      A     M   1503.7;
      A     M    184.1;
      A     M   1606.6;
      A     M   1600.0;
      O     ;
      A     M   1503.5;
      A     M    184.0;
      A(    ;
      O     M   1707.0;
      O     ;
      A     M   1702.0;
      A     M   1702.2;
      A     M   1702.4;
      A     M   1702.6;
      A     M   1703.0;
      A     M   1703.2;
      A     M   1703.4;
      A     M   1703.6;
      A     M   1706.7;
      A     M   1704.0;
      A     M   1704.2;
      A     M   1704.5;
      A     M   1704.6;
      )     ;
      A     M   1706.1;
      A     M   1701.0;
      =     Q   1058.0;
NETWORK
TITLE =

      A     M   4108.1;
      =     Q   1058.1;
NETWORK
TITLE =

      A     M   1503.7;
      A     M    184.1;
      A     M   1606.6;
      A     M   1600.0;
      =     Q   1059.0;
NETWORK
TITLE =

      A     M   1503.5;
      A     M    184.0;
      A     M   1701.0;
      A     M   1706.1;
      A(    ;
      O     M   1707.0;
      O     ;
      A     M   1702.0;
      A     M   1702.2;
      A     M   1702.4;
      A     M   1702.6;
      A     M   1703.0;
      A     M   1703.2;
      A     M   1703.4;
      A     M   1703.6;
      A     M   1706.7;
      A     M   1704.0;
      A     M   1704.2;
      A     M   1704.5;
      A     M   1704.6;
      )     ;
      =     Q   1059.2;
END_FUNCTION

FUNCTION FC 137 : VOID
TITLE =
VERSION : 0.1

BEGIN
NETWORK
TITLE =
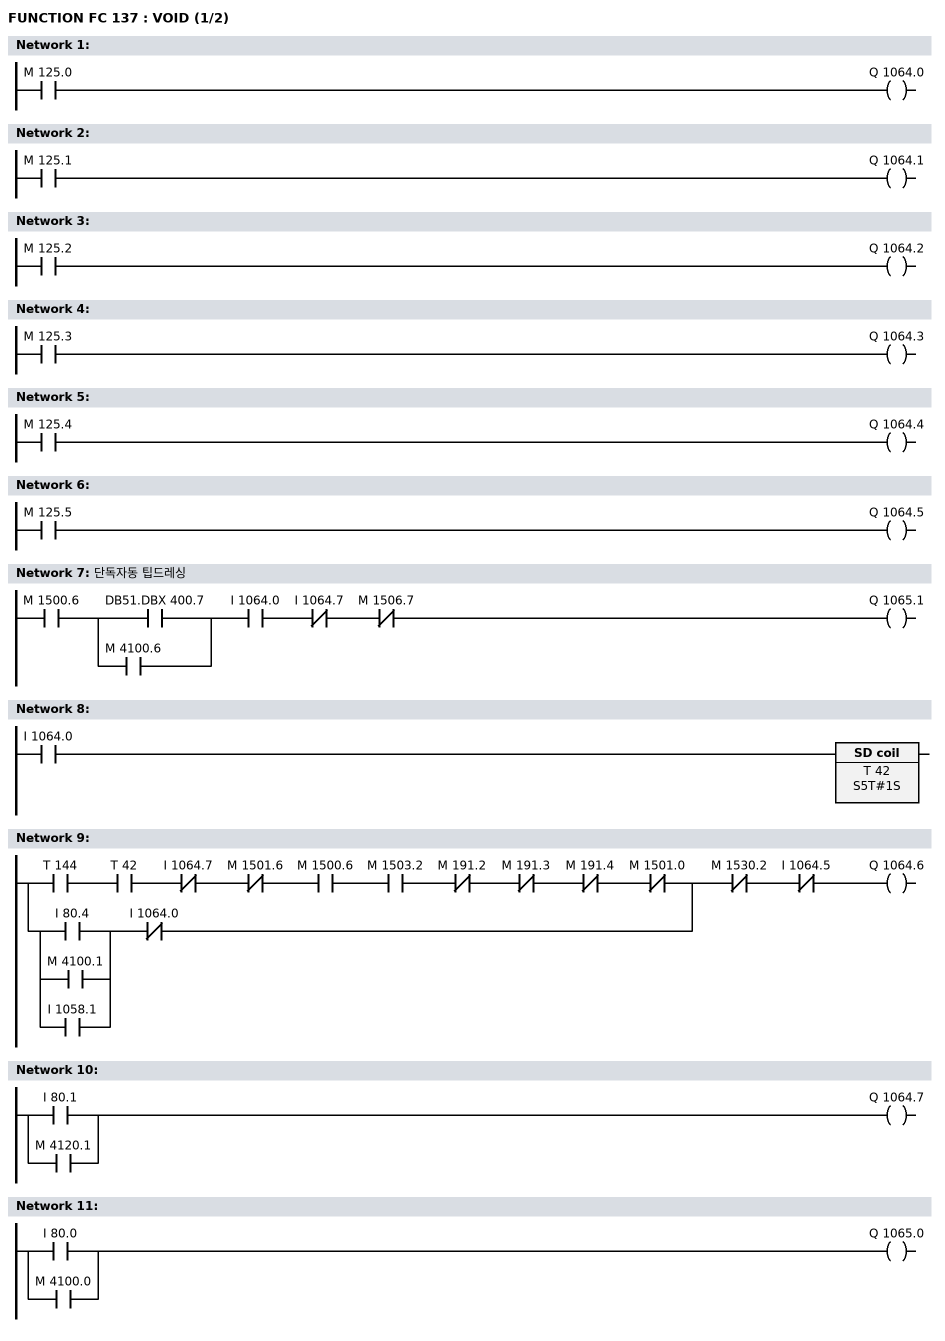

      A     M    125.0;
      =     Q   1064.0;
NETWORK
TITLE =

      A     M    125.1;
      =     Q   1064.1;
NETWORK
TITLE =

      A     M    125.2;
      =     Q   1064.2;
NETWORK
TITLE =

      A     M    125.3;
      =     Q   1064.3;
NETWORK
TITLE =

      A     M    125.4;
      =     Q   1064.4;
NETWORK
TITLE =

      A     M    125.5;
      =     Q   1064.5;
NETWORK
TITLE =단독자동 팁드레싱

      A     M   1500.6;
      A(    ;
      O     DB51.DBX  400.7;
      O     M   4100.6;
      )     ;
      A     I   1064.0;
      AN    I   1064.7;
      AN    M   1506.7;
      =     Q   1065.1;
NETWORK
TITLE =

      A     I   1064.0;
      L     S5T#1S;
      SD    T     42;
NETWORK
TITLE =

      A(    ;
      A     T    144;
      A     T     42;
      AN    I   1064.7;
      AN    M   1501.6;
      A     M   1500.6;
      A     M   1503.2;
      AN    M    191.2;
      AN    M    191.3;
      AN    M    191.4;
      AN    M   1501.0;
      O     ;
      A(    ;
      O     I     80.4;
      O     M   4100.1;
      O     I   1058.1;
      )     ;
      AN    I   1064.0;
      )     ;
      AN    M   1530.2;
      AN    I   1064.5;
      =     Q   1064.6;
NETWORK
TITLE =

      O     I     80.1;
      O     M   4120.1;
      =     Q   1064.7;
NETWORK
TITLE =

      O     I     80.0;
      O     M   4100.0;
      =     Q   1065.0;
NETWORK
TITLE =
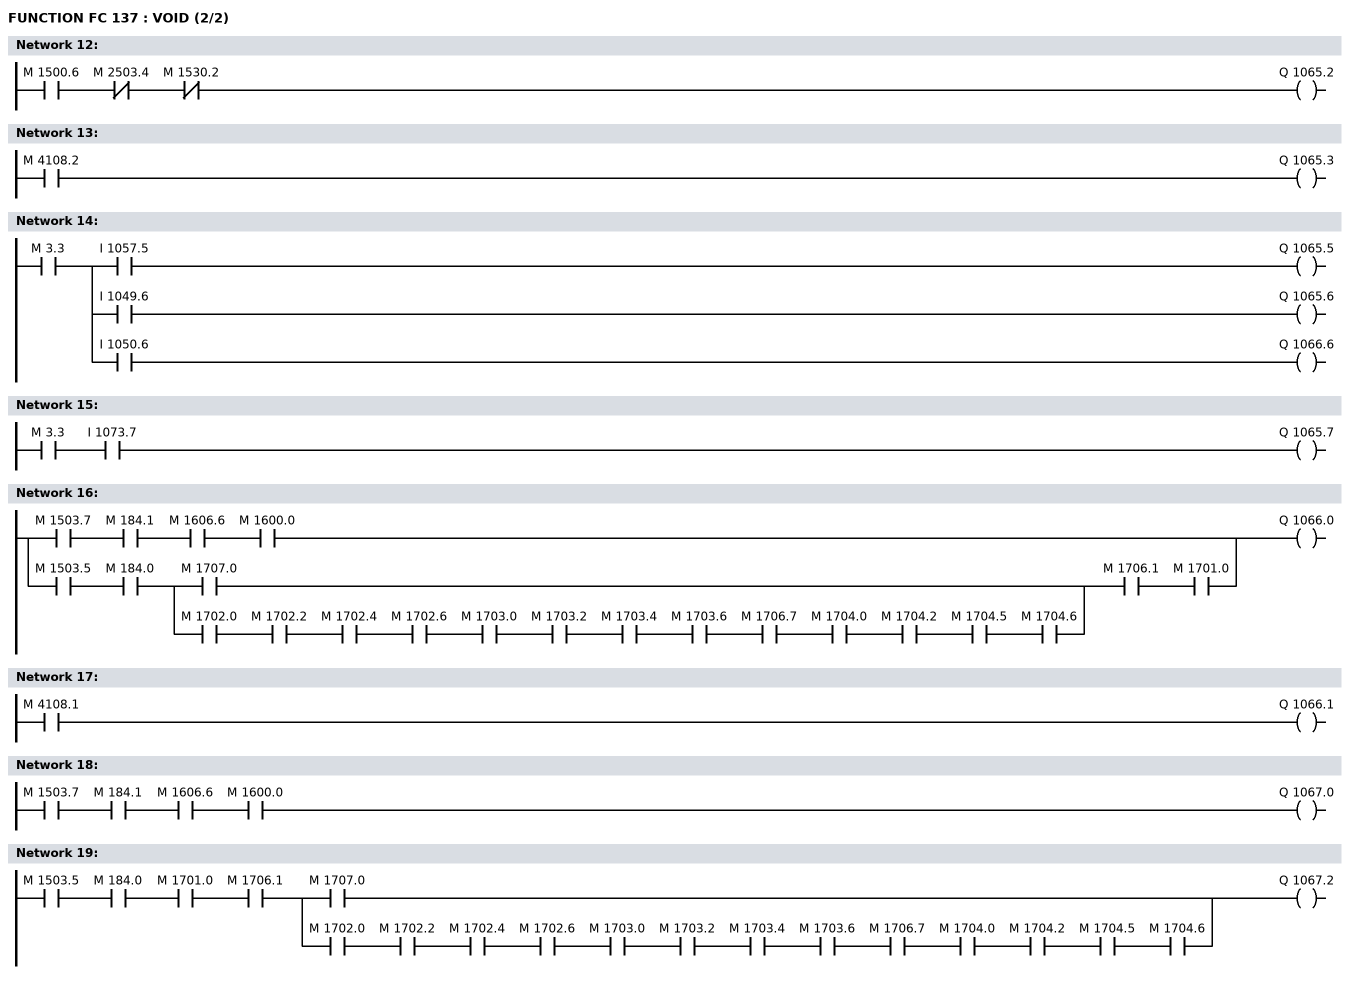

      A     M   1500.6;
      AN    M   2503.4;
      AN    M   1530.2;
      =     Q   1065.2;
NETWORK
TITLE =

      A     M   4108.2;
      =     Q   1065.3;
NETWORK
TITLE =

      A     M      3.3;
      =     L      0.0;
      A     L      0.0;
      A     I   1057.5;
      =     Q   1065.5;
      A     L      0.0;
      A     I   1049.6;
      =     Q   1065.6;
      A     L      0.0;
      A     I   1050.6;
      =     Q   1066.6;
NETWORK
TITLE =

      A     M      3.3;
      A     I   1073.7;
      =     Q   1065.7;
NETWORK
TITLE =

      A     M   1503.7;
      A     M    184.1;
      A     M   1606.6;
      A     M   1600.0;
      O     ;
      A     M   1503.5;
      A     M    184.0;
      A(    ;
      O     M   1707.0;
      O     ;
      A     M   1702.0;
      A     M   1702.2;
      A     M   1702.4;
      A     M   1702.6;
      A     M   1703.0;
      A     M   1703.2;
      A     M   1703.4;
      A     M   1703.6;
      A     M   1706.7;
      A     M   1704.0;
      A     M   1704.2;
      A     M   1704.5;
      A     M   1704.6;
      )     ;
      A     M   1706.1;
      A     M   1701.0;
      =     Q   1066.0;
NETWORK
TITLE =

      A     M   4108.1;
      =     Q   1066.1;
NETWORK
TITLE =

      A     M   1503.7;
      A     M    184.1;
      A     M   1606.6;
      A     M   1600.0;
      =     Q   1067.0;
NETWORK
TITLE =

      A     M   1503.5;
      A     M    184.0;
      A     M   1701.0;
      A     M   1706.1;
      A(    ;
      O     M   1707.0;
      O     ;
      A     M   1702.0;
      A     M   1702.2;
      A     M   1702.4;
      A     M   1702.6;
      A     M   1703.0;
      A     M   1703.2;
      A     M   1703.4;
      A     M   1703.6;
      A     M   1706.7;
      A     M   1704.0;
      A     M   1704.2;
      A     M   1704.5;
      A     M   1704.6;
      )     ;
      =     Q   1067.2;
END_FUNCTION

FUNCTION FC 138 : VOID
TITLE =
VERSION : 0.1

BEGIN
NETWORK
TITLE =
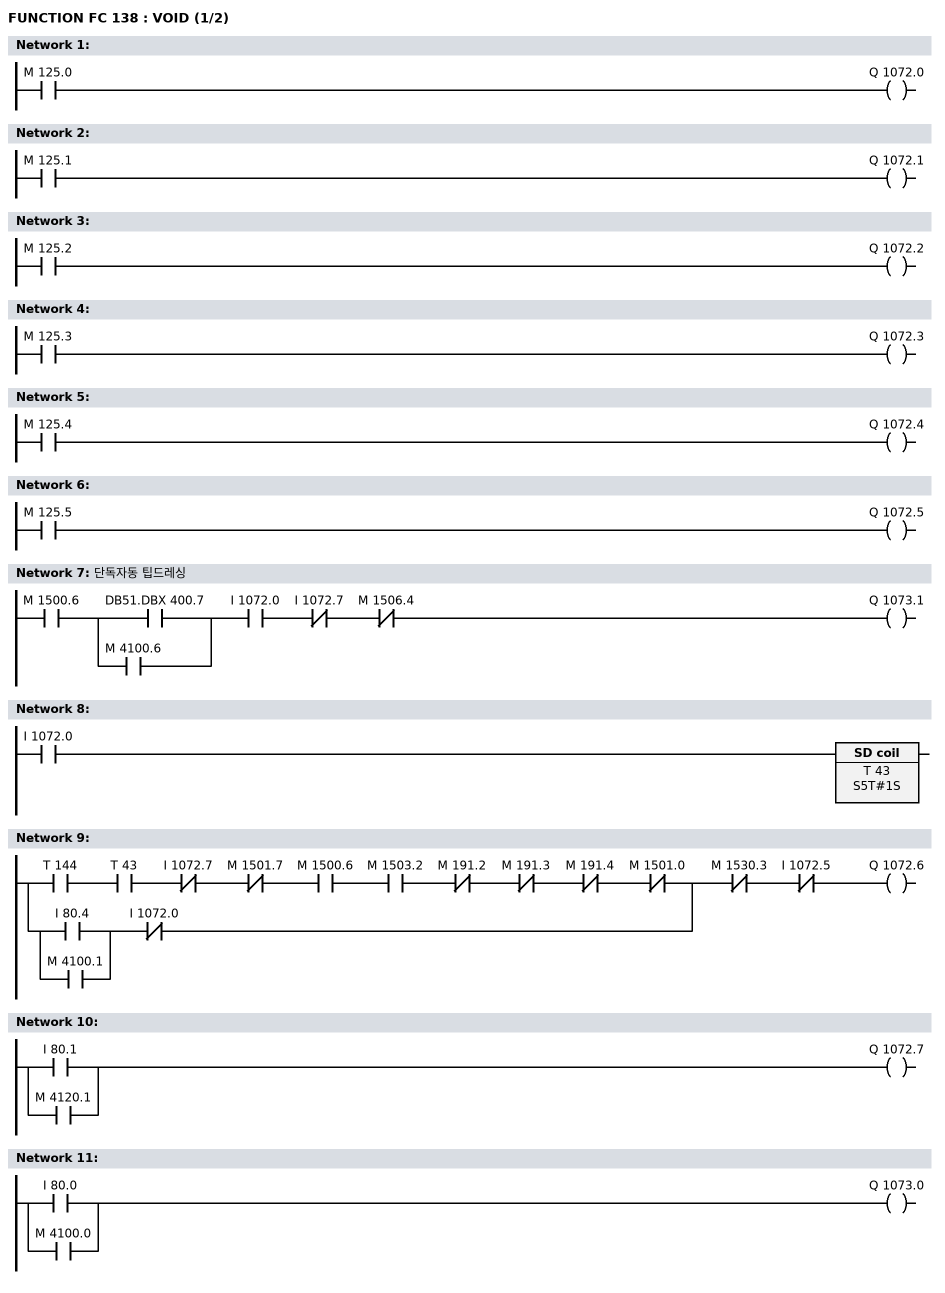

      A     M    125.0;
      =     Q   1072.0;
NETWORK
TITLE =

      A     M    125.1;
      =     Q   1072.1;
NETWORK
TITLE =

      A     M    125.2;
      =     Q   1072.2;
NETWORK
TITLE =

      A     M    125.3;
      =     Q   1072.3;
NETWORK
TITLE =

      A     M    125.4;
      =     Q   1072.4;
NETWORK
TITLE =

      A     M    125.5;
      =     Q   1072.5;
NETWORK
TITLE =단독자동 팁드레싱

      A     M   1500.6;
      A(    ;
      O     DB51.DBX  400.7;
      O     M   4100.6;
      )     ;
      A     I   1072.0;
      AN    I   1072.7;
      AN    M   1506.4;
      =     Q   1073.1;
NETWORK
TITLE =

      A     I   1072.0;
      L     S5T#1S;
      SD    T     43;
NETWORK
TITLE =

      A(    ;
      A     T    144;
      A     T     43;
      AN    I   1072.7;
      AN    M   1501.7;
      A     M   1500.6;
      A     M   1503.2;
      AN    M    191.2;
      AN    M    191.3;
      AN    M    191.4;
      AN    M   1501.0;
      O     ;
      A(    ;
      O     I     80.4;
      O     M   4100.1;
      )     ;
      AN    I   1072.0;
      )     ;
      AN    M   1530.3;
      AN    I   1072.5;
      =     Q   1072.6;
NETWORK
TITLE =

      O     I     80.1;
      O     M   4120.1;
      =     Q   1072.7;
NETWORK
TITLE =

      O     I     80.0;
      O     M   4100.0;
      =     Q   1073.0;
NETWORK
TITLE =
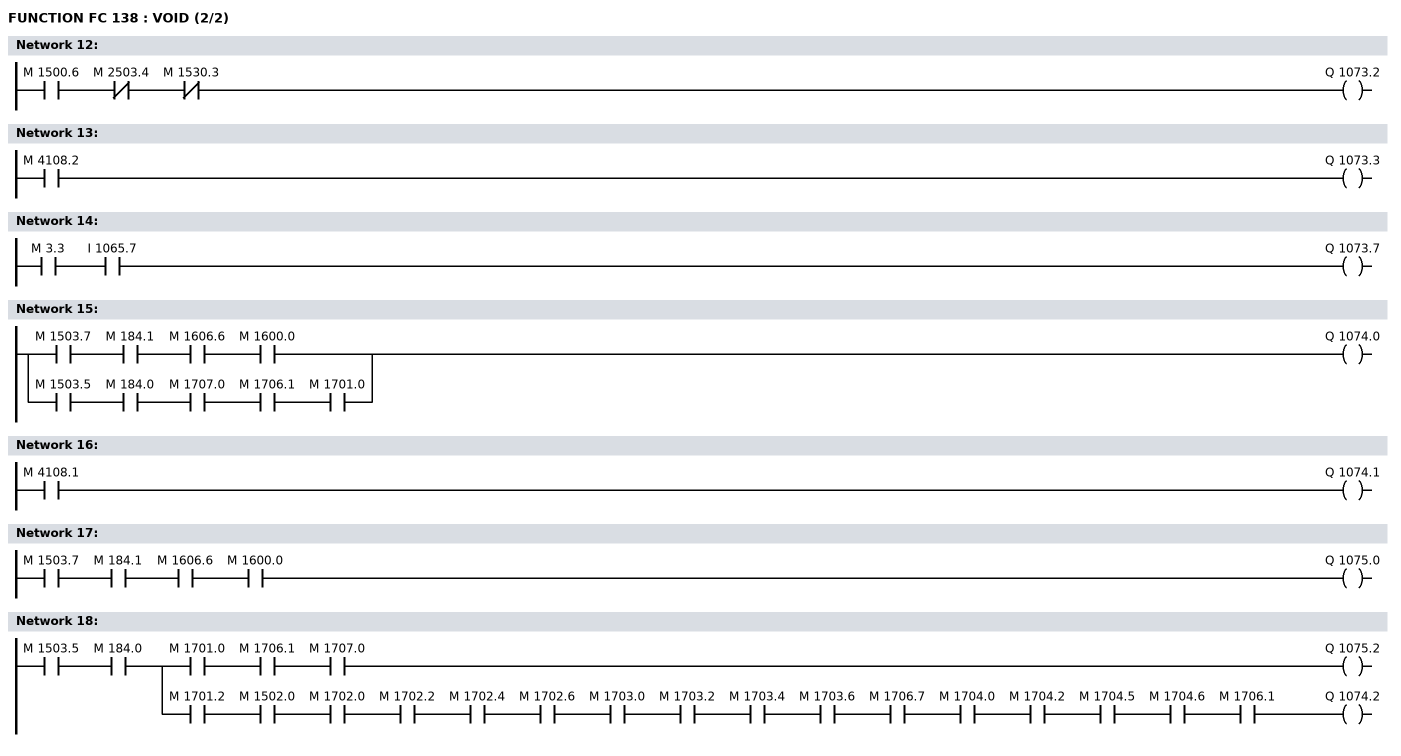

      A     M   1500.6;
      AN    M   2503.4;
      AN    M   1530.3;
      =     Q   1073.2;
NETWORK
TITLE =

      A     M   4108.2;
      =     Q   1073.3;
NETWORK
TITLE =

      A     M      3.3;
      A     I   1065.7;
      =     Q   1073.7;
NETWORK
TITLE =

      A     M   1503.7;
      A     M    184.1;
      A     M   1606.6;
      A     M   1600.0;
      O     ;
      A     M   1503.5;
      A     M    184.0;
      A     M   1707.0;
      A     M   1706.1;
      A     M   1701.0;
      =     Q   1074.0;
NETWORK
TITLE =

      A     M   4108.1;
      =     Q   1074.1;
NETWORK
TITLE =

      A     M   1503.7;
      A     M    184.1;
      A     M   1606.6;
      A     M   1600.0;
      =     Q   1075.0;
NETWORK
TITLE =

      A     M   1503.5;
      A     M    184.0;
      =     L      0.0;
      A     L      0.0;
      A     M   1701.0;
      A     M   1706.1;
      A     M   1707.0;
      =     Q   1075.2;
      A     L      0.0;
      A     M   1701.2;
      A     M   1502.0;
      A     M   1702.0;
      A     M   1702.2;
      A     M   1702.4;
      A     M   1702.6;
      A     M   1703.0;
      A     M   1703.2;
      A     M   1703.4;
      A     M   1703.6;
      A     M   1706.7;
      A     M   1704.0;
      A     M   1704.2;
      A     M   1704.5;
      A     M   1704.6;
      A     M   1706.1;
      =     Q   1074.2;
END_FUNCTION

FUNCTION_BLOCK FB 140
TITLE =
VERSION : 0.1


VAR
  S708_MODE : FB 402;
END_VAR
BEGIN
NETWORK
TITLE =
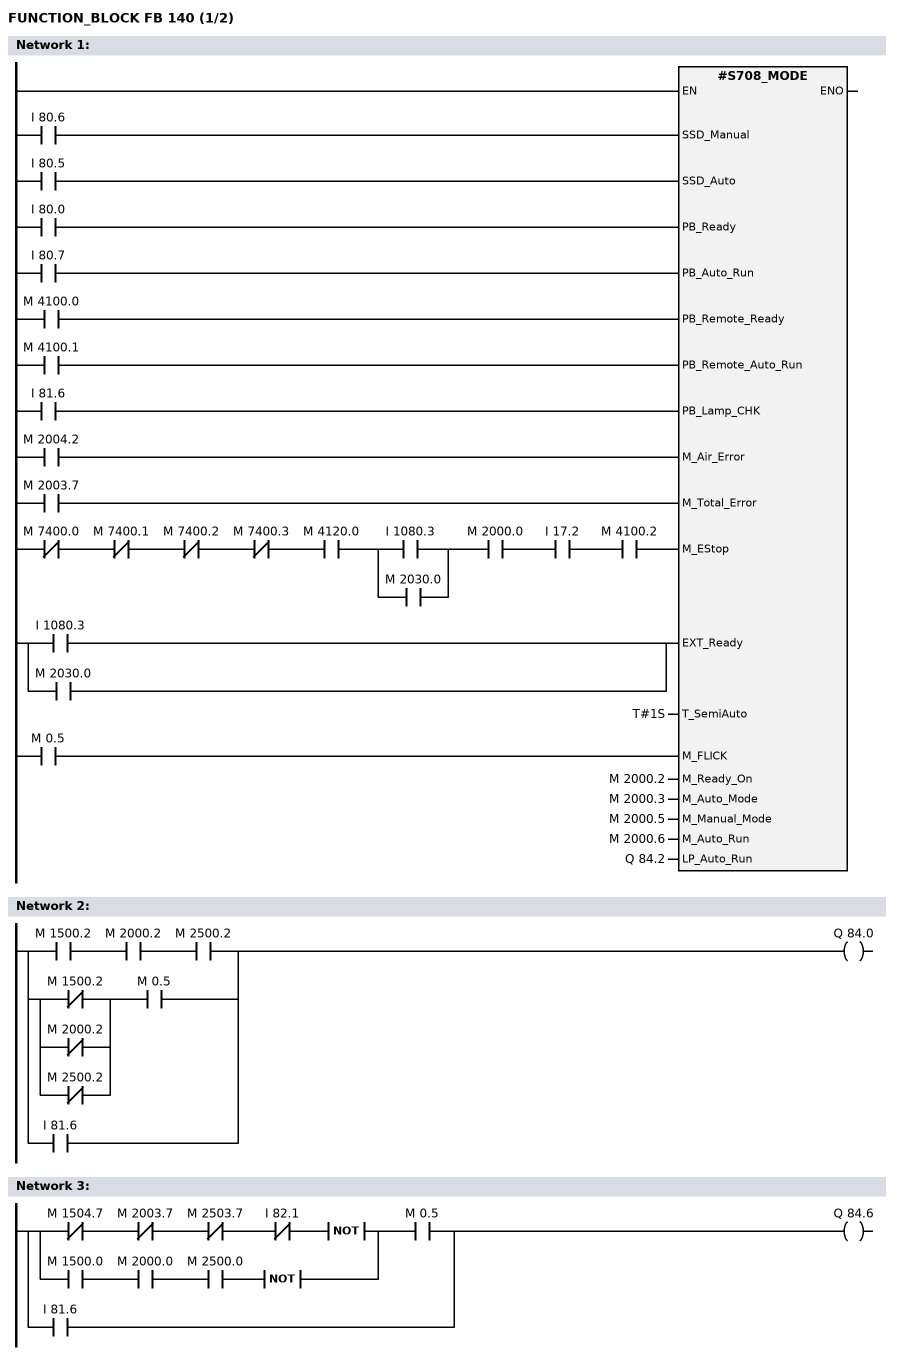

      A     I     80.6;
      =     L      0.0;
      BLD   103;
      A     I     80.5;
      =     L      0.1;
      BLD   103;
      A     I     80.0;
      =     L      0.2;
      BLD   103;
      A     I     80.7;
      =     L      0.3;
      BLD   103;
      A     M   4100.0;
      =     L      0.4;
      BLD   103;
      A     M   4100.1;
      =     L      0.5;
      BLD   103;
      A     I     81.6;
      =     L      0.6;
      BLD   103;
      A     M   2004.2;
      =     L      0.7;
      BLD   103;
      A     M   2003.7;
      =     L      1.1;
      BLD   103;
      AN    M   7400.0;
      AN    M   7400.1;
      AN    M   7400.2;
      AN    M   7400.3;
      A     M   4120.0;
      A(    ;
      O     I   1080.3;
      O     M   2030.0;
      )     ;
      A     M   2000.0;
      A     I     17.2;
      A     M   4100.2;
      =     L      1.2;
      BLD   103;
      A(    ;
      O     I   1080.3;
      O     M   2030.0;
      )     ;
      =     L      1.3;
      BLD   103;
      A     M      0.5;
      =     L      1.5;
      BLD   103;
      CALL #S708_MODE (
           SSD_Manual               := L      0.0,
           SSD_Auto                 := L      0.1,
           PB_Ready                 := L      0.2,
           PB_Auto_Run              := L      0.3,
           PB_Remote_Ready          := L      0.4,
           PB_Remote_Auto_Run       := L      0.5,
           PB_Lamp_CHK              := L      0.6,
           M_Air_Error              := L      0.7,
           M_Total_Error            := L      1.1,
           M_EStop                  := L      1.2,
           EXT_Ready                := L      1.3,
           T_SemiAuto               := T#1S,
           M_FLICK                  := L      1.5,
           M_Ready_On               := M   2000.2,
           M_Auto_Mode              := M   2000.3,
           M_Manual_Mode            := M   2000.5,
           M_Auto_Run               := M   2000.6,
           LP_Auto_Run              := Q     84.2);
      NOP   0;
NETWORK
TITLE =

      A     M   1500.2;
      A     M   2000.2;
      A     M   2500.2;
      O     ;
      A(    ;
      ON    M   1500.2;
      ON    M   2000.2;
      ON    M   2500.2;
      )     ;
      A     M      0.5;
      O     I     81.6;
      =     Q     84.0;
NETWORK
TITLE =

      A(    ;
      AN    M   1504.7;
      AN    M   2003.7;
      AN    M   2503.7;
      AN    I     82.1;
      NOT   ;
      O(    ;
      A     M   1500.0;
      A     M   2000.0;
      A     M   2500.0;
      NOT   ;
      )     ;
      )     ;
      A     M      0.5;
      O     I     81.6;
      =     Q     84.6;
NETWORK
TITLE =
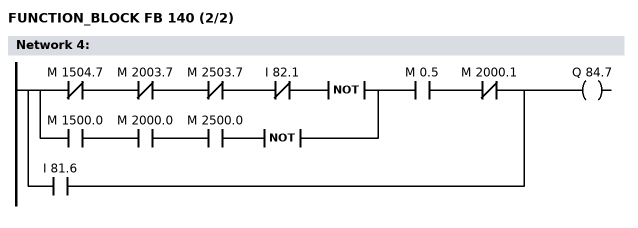

      A(    ;
      AN    M   1504.7;
      AN    M   2003.7;
      AN    M   2503.7;
      AN    I     82.1;
      NOT   ;
      O(    ;
      A     M   1500.0;
      A     M   2000.0;
      A     M   2500.0;
      NOT   ;
      )     ;
      )     ;
      A     M      0.5;
      AN    M   2000.1;
      O     I     81.6;
      =     Q     84.7;
END_FUNCTION_BLOCK

DATA_BLOCK DB 140
TITLE =
VERSION : 0.0

 FB 140
BEGIN
   S708_MODE.SSD_Manual := FALSE;
   S708_MODE.SSD_Auto := TRUE;
   S708_MODE.PB_Ready := FALSE;
   S708_MODE.PB_Auto_Run := FALSE;
   S708_MODE.PB_Remote_Ready := FALSE;
   S708_MODE.PB_Remote_Auto_Run := FALSE;
   S708_MODE.PB_Lamp_CHK := FALSE;
   S708_MODE.M_Air_Error := FALSE;
   S708_MODE.M_Water_Error := FALSE;
   S708_MODE.M_Total_Error := FALSE;
   S708_MODE.M_EStop := TRUE;
   S708_MODE.EXT_Ready := TRUE;
   S708_MODE.EXT_Auto := FALSE;
   S708_MODE.T_SemiAuto := T#1S;
   S708_MODE.M_FLICK := TRUE;
   S708_MODE.M_Ready_On := TRUE;
   S708_MODE.M_Auto_Mode := TRUE;
   S708_MODE.M_SemiAuto_Mode := FALSE;
   S708_MODE.M_Manual_Mode := FALSE;
   S708_MODE.M_Auto_Run := TRUE;
   S708_MODE.LP_Ready_On := TRUE;
   S708_MODE.LP_Auto_Run := TRUE;
   S708_MODE.AUTO_MODE_DELAY.IN := FALSE;
   S708_MODE.AUTO_MODE_DELAY.PT := T#0MS;
   S708_MODE.AUTO_MODE_DELAY.Q := FALSE;
   S708_MODE.AUTO_MODE_DELAY.ET := T#0MS;
   S708_MODE.AUTO_MODE_DELAY.STATE := B#16#0;
   S708_MODE.AUTO_MODE_DELAY.STIME := T#0MS;
   S708_MODE.AUTO_MODE_DELAY.ATIME := T#0MS;
   S708_MODE.SEMI_AUTO_DELAY.IN := FALSE;
   S708_MODE.SEMI_AUTO_DELAY.PT := T#1S;
   S708_MODE.SEMI_AUTO_DELAY.Q := FALSE;
   S708_MODE.SEMI_AUTO_DELAY.ET := T#0MS;
   S708_MODE.SEMI_AUTO_DELAY.STATE := B#16#0;
   S708_MODE.SEMI_AUTO_DELAY.STIME := T#21D23H22M46S522MS;
   S708_MODE.SEMI_AUTO_DELAY.ATIME := T#21D23H22M46S547MS;
   S708_MODE.MANUAL_DELAY.IN := FALSE;
   S708_MODE.MANUAL_DELAY.PT := T#0MS;
   S708_MODE.MANUAL_DELAY.Q := FALSE;
   S708_MODE.MANUAL_DELAY.ET := T#0MS;
   S708_MODE.MANUAL_DELAY.STATE := B#16#0;
   S708_MODE.MANUAL_DELAY.STIME := T#0MS;
   S708_MODE.MANUAL_DELAY.ATIME := T#0MS;
END_DATA_BLOCK

FUNCTION FC 140 : VOID
TITLE =
VERSION : 0.1

BEGIN
NETWORK
TITLE =
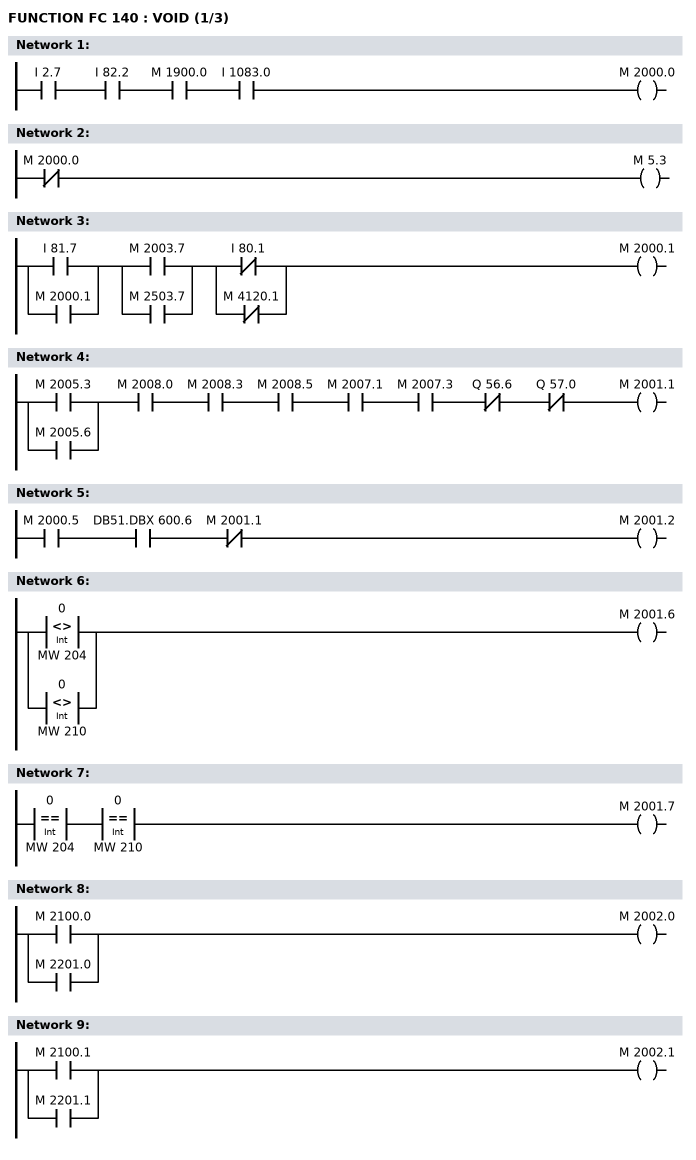

      A     I      2.7;
      A     I     82.2;
      A     M   1900.0;
      A     I   1083.0;
      =     M   2000.0;
NETWORK
TITLE =

      AN    M   2000.0;
      =     M      5.3;
NETWORK
TITLE =

      A(    ;
      O     I     81.7;
      O     M   2000.1;
      )     ;
      A(    ;
      O     M   2003.7;
      O     M   2503.7;
      )     ;
      A(    ;
      ON    I     80.1;
      ON    M   4120.1;
      )     ;
      =     M   2000.1;
NETWORK
TITLE =

      A(    ;
      O     M   2005.3;
      O     M   2005.6;
      )     ;
      A     M   2008.0;
      A     M   2008.3;
      A     M   2008.5;
      A     M   2007.1;
      A     M   2007.3;
      AN    Q     56.6;
      AN    Q     57.0;
      =     M   2001.1;
NETWORK
TITLE =

      A     M   2000.5;
      A     DB51.DBX  600.6;
      AN    M   2001.1;
      =     M   2001.2;
NETWORK
TITLE =

      O(    ;
      L     0;
      L     MW   204;
      <>I   ;
      )     ;
      O(    ;
      L     0;
      L     MW   210;
      <>I   ;
      )     ;
      =     M   2001.6;
NETWORK
TITLE =

      A(    ;
      L     0;
      L     MW   204;
      ==I   ;
      )     ;
      A(    ;
      L     0;
      L     MW   210;
      ==I   ;
      )     ;
      =     M   2001.7;
NETWORK
TITLE =

      O     M   2100.0;
      O     M   2201.0;
      =     M   2002.0;
NETWORK
TITLE =

      O     M   2100.1;
      O     M   2201.1;
      =     M   2002.1;
NETWORK
TITLE =
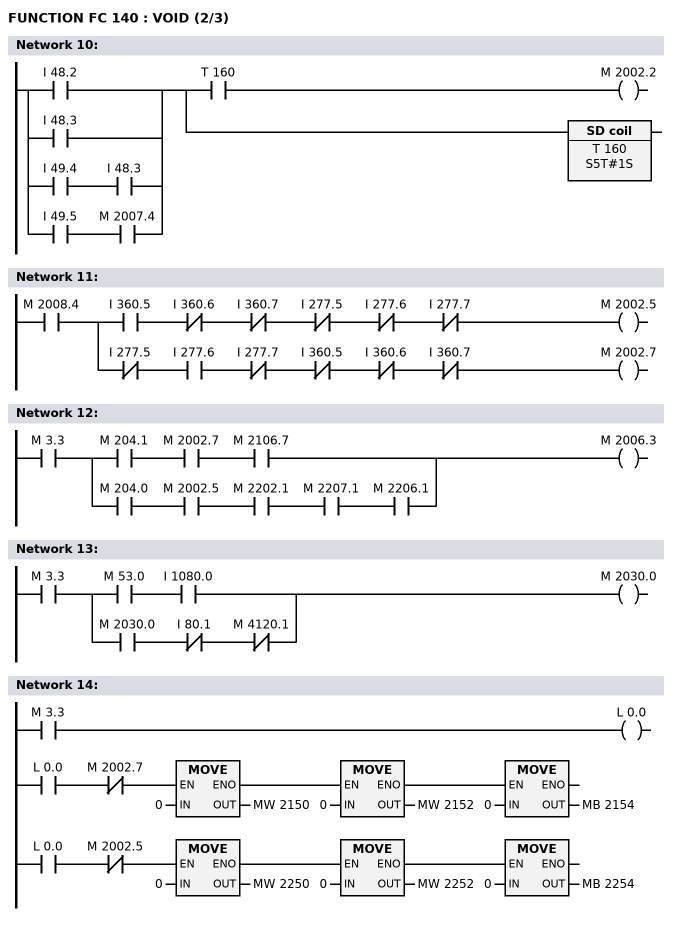

      O     I     48.2;
      O     I     48.3;
      O     ;
      A     I     49.4;
      A     I     48.3;
      O     ;
      A     I     49.5;
      A     M   2007.4;
      =     L      0.0;
      A     L      0.0;
      A     T    160;
      =     M   2002.2;
      A     L      0.0;
      BLD   102;
      L     S5T#1S;
      SD    T    160;
NETWORK
TITLE =

      A     M   2008.4;
      =     L      0.0;
      A     L      0.0;
      A     I    360.5;
      AN    I    360.6;
      AN    I    360.7;
      AN    I    277.5;
      AN    I    277.6;
      AN    I    277.7;
      =     M   2002.5;
      A     L      0.0;
      AN    I    277.5;
      A     I    277.6;
      AN    I    277.7;
      AN    I    360.5;
      AN    I    360.6;
      AN    I    360.7;
      =     M   2002.7;
NETWORK
TITLE =

      A     M      3.3;
      A(    ;
      A     M    204.1;
      A     M   2002.7;
      A     M   2106.7;
      O     ;
      A     M    204.0;
      A     M   2002.5;
      A     M   2202.1;
      A     M   2207.1;
      A     M   2206.1;
      )     ;
      =     M   2006.3;
NETWORK
TITLE =

      A     M      3.3;
      A(    ;
      A     M     53.0;
      A     I   1080.0;
      O     ;
      A     M   2030.0;
      AN    I     80.1;
      AN    M   4120.1;
      )     ;
      =     M   2030.0;
NETWORK
TITLE =

      A     M      3.3;
      =     L      0.0;
      A(    ;
      A(    ;
      A     L      0.0;
      AN    M   2002.7;
      JNB   _001;
      L     0;
      T     MW  2150;
      SET   ;
      SAVE  ;
      CLR   ;
_001: A     BR;
      )     ;
      JNB   _002;
      L     0;
      T     MW  2152;
      SET   ;
      SAVE  ;
      CLR   ;
_002: A     BR;
      )     ;
      JNB   _003;
      L     0;
      T     MB  2154;
_003: NOP   0;
      A(    ;
      A(    ;
      A     L      0.0;
      AN    M   2002.5;
      JNB   _004;
      L     0;
      T     MW  2250;
      SET   ;
      SAVE  ;
      CLR   ;
_004: A     BR;
      )     ;
      JNB   _005;
      L     0;
      T     MW  2252;
      SET   ;
      SAVE  ;
      CLR   ;
_005: A     BR;
      )     ;
      JNB   _006;
      L     0;
      T     MB  2254;
_006: NOP   0;
NETWORK
TITLE =
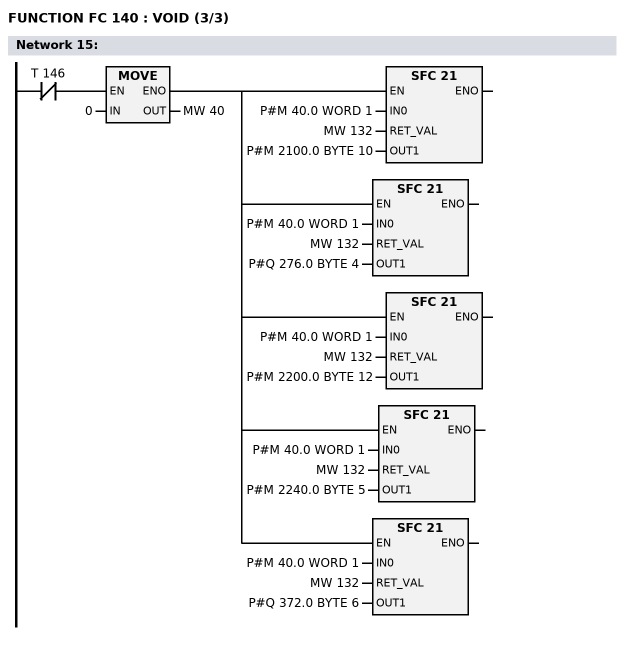

      AN    T    146;
      JNB   _007;
      L     0;
      T     MW    40;
      SET   ;
      SAVE  ;
      CLR   ;
_007: A     BR;
      =     L      0.0;
      A     L      0.0;
      JNB   _008;
      CALL SFC   21 (
           IN0                      := P#M 40.0 WORD 1,
           RET_VAL                  := MW   132,
           OUT1                     := P#M 2100.0 BYTE 10);
_008: NOP   0;
      A     L      0.0;
      JNB   _009;
      CALL SFC   21 (
           IN0                      := P#M 40.0 WORD 1,
           RET_VAL                  := MW   132,
           OUT1                     := P#Q 276.0 BYTE 4);
_009: NOP   0;
      A     L      0.0;
      JNB   _00a;
      CALL SFC   21 (
           IN0                      := P#M 40.0 WORD 1,
           RET_VAL                  := MW   132,
           OUT1                     := P#M 2200.0 BYTE 12);
_00a: NOP   0;
      A     L      0.0;
      JNB   _00b;
      CALL SFC   21 (
           IN0                      := P#M 40.0 WORD 1,
           RET_VAL                  := MW   132,
           OUT1                     := P#M 2240.0 BYTE 5);
_00b: NOP   0;
      A     L      0.0;
      JNB   _00c;
      CALL SFC   21 (
           IN0                      := P#M 40.0 WORD 1,
           RET_VAL                  := MW   132,
           OUT1                     := P#Q 372.0 BYTE 6);
_00c: NOP   0;
END_FUNCTION

FUNCTION_BLOCK FB 141
TITLE =
VERSION : 0.1


VAR
  S708_HOOK_PIN : FB 424;
  S708_EJECT : FB 424;
  S708_SAFETY_PIN : FB 424;
  S708_ELE_UP_DN : FB 424;
  S708_ELE_ADV_RET : FB 424;
  S708_AIR_ELE_ADV_RET : FB 424;
END_VAR
BEGIN
NETWORK
TITLE =
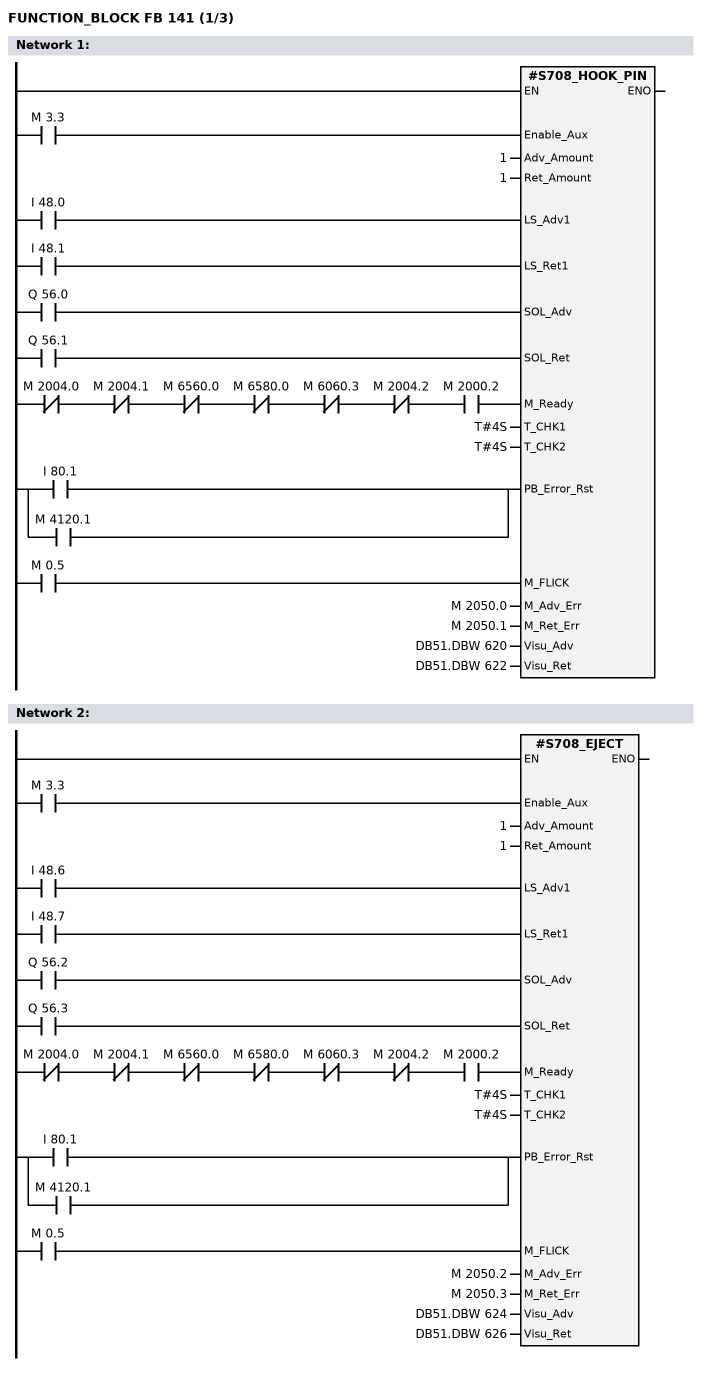

      A     M      3.3;
      =     L      0.0;
      BLD   103;
      A     I     48.0;
      =     L      0.1;
      BLD   103;
      A     I     48.1;
      =     L      0.2;
      BLD   103;
      A     Q     56.0;
      =     L      1.1;
      BLD   103;
      A     Q     56.1;
      =     L      1.2;
      BLD   103;
      AN    M   2004.0;
      AN    M   2004.1;
      AN    M   6560.0;
      AN    M   6580.0;
      AN    M   6060.3;
      AN    M   2004.2;
      A     M   2000.2;
      =     L      1.3;
      BLD   103;
      A(    ;
      O     I     80.1;
      O     M   4120.1;
      )     ;
      =     L      1.5;
      BLD   103;
      A     M      0.5;
      =     L      1.6;
      BLD   103;
      CALL #S708_HOOK_PIN (
           Enable_Aux               := L      0.0,
           Adv_Amount               := 1,
           Ret_Amount               := 1,
           LS_Adv1                  := L      0.1,
           LS_Ret1                  := L      0.2,
           SOL_Adv                  := L      1.1,
           SOL_Ret                  := L      1.2,
           M_Ready                  := L      1.3,
           T_CHK1                   := T#4S,
           T_CHK2                   := T#4S,
           PB_Error_Rst             := L      1.5,
           M_FLICK                  := L      1.6,
           M_Adv_Err                := M   2050.0,
           M_Ret_Err                := M   2050.1,
           Visu_Adv                 := DB51.DBW  620,
           Visu_Ret                 := DB51.DBW  622);
      NOP   0;
NETWORK
TITLE =

      A     M      3.3;
      =     L      0.0;
      BLD   103;
      A     I     48.6;
      =     L      0.1;
      BLD   103;
      A     I     48.7;
      =     L      0.2;
      BLD   103;
      A     Q     56.2;
      =     L      1.1;
      BLD   103;
      A     Q     56.3;
      =     L      1.2;
      BLD   103;
      AN    M   2004.0;
      AN    M   2004.1;
      AN    M   6560.0;
      AN    M   6580.0;
      AN    M   6060.3;
      AN    M   2004.2;
      A     M   2000.2;
      =     L      1.3;
      BLD   103;
      A(    ;
      O     I     80.1;
      O     M   4120.1;
      )     ;
      =     L      1.5;
      BLD   103;
      A     M      0.5;
      =     L      1.6;
      BLD   103;
      CALL #S708_EJECT (
           Enable_Aux               := L      0.0,
           Adv_Amount               := 1,
           Ret_Amount               := 1,
           LS_Adv1                  := L      0.1,
           LS_Ret1                  := L      0.2,
           SOL_Adv                  := L      1.1,
           SOL_Ret                  := L      1.2,
           M_Ready                  := L      1.3,
           T_CHK1                   := T#4S,
           T_CHK2                   := T#4S,
           PB_Error_Rst             := L      1.5,
           M_FLICK                  := L      1.6,
           M_Adv_Err                := M   2050.2,
           M_Ret_Err                := M   2050.3,
           Visu_Adv                 := DB51.DBW  624,
           Visu_Ret                 := DB51.DBW  626);
      NOP   0;
NETWORK
TITLE =
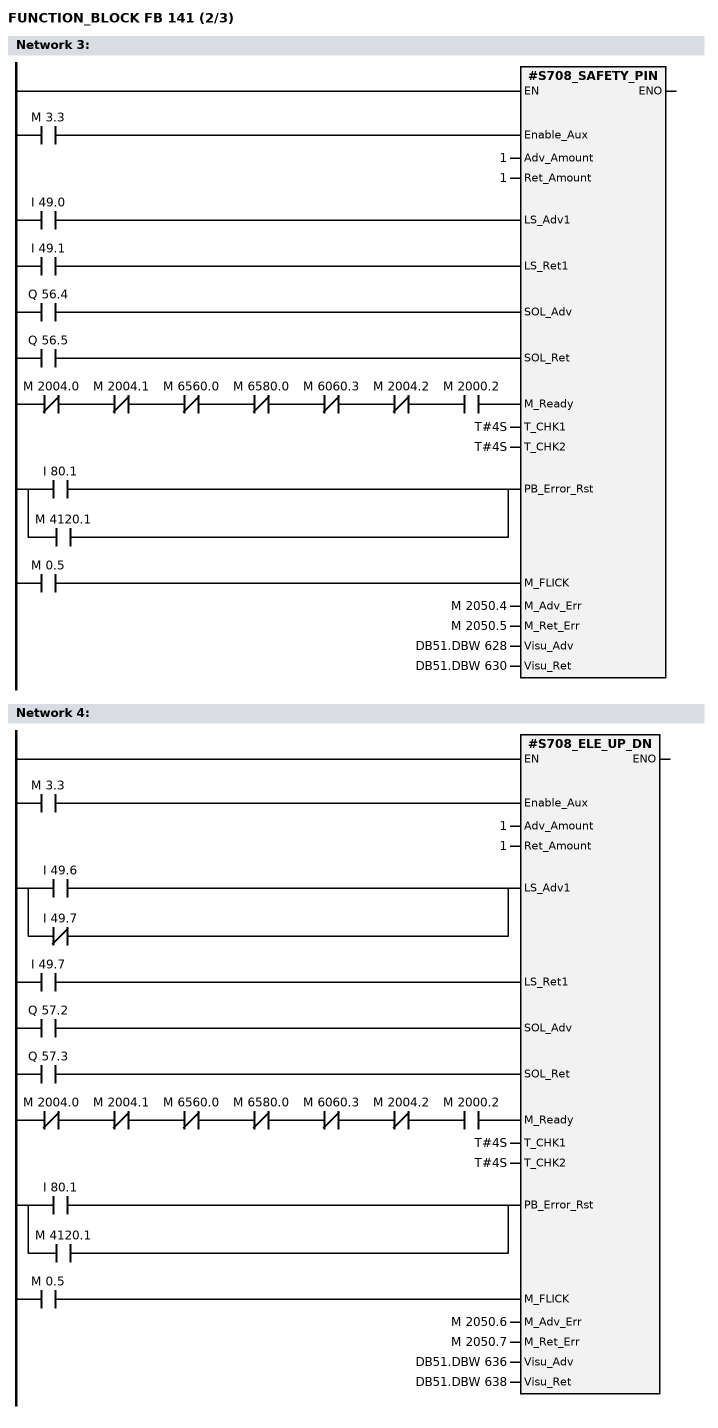

      A     M      3.3;
      =     L      0.0;
      BLD   103;
      A     I     49.0;
      =     L      0.1;
      BLD   103;
      A     I     49.1;
      =     L      0.2;
      BLD   103;
      A     Q     56.4;
      =     L      1.1;
      BLD   103;
      A     Q     56.5;
      =     L      1.2;
      BLD   103;
      AN    M   2004.0;
      AN    M   2004.1;
      AN    M   6560.0;
      AN    M   6580.0;
      AN    M   6060.3;
      AN    M   2004.2;
      A     M   2000.2;
      =     L      1.3;
      BLD   103;
      A(    ;
      O     I     80.1;
      O     M   4120.1;
      )     ;
      =     L      1.5;
      BLD   103;
      A     M      0.5;
      =     L      1.6;
      BLD   103;
      CALL #S708_SAFETY_PIN (
           Enable_Aux               := L      0.0,
           Adv_Amount               := 1,
           Ret_Amount               := 1,
           LS_Adv1                  := L      0.1,
           LS_Ret1                  := L      0.2,
           SOL_Adv                  := L      1.1,
           SOL_Ret                  := L      1.2,
           M_Ready                  := L      1.3,
           T_CHK1                   := T#4S,
           T_CHK2                   := T#4S,
           PB_Error_Rst             := L      1.5,
           M_FLICK                  := L      1.6,
           M_Adv_Err                := M   2050.4,
           M_Ret_Err                := M   2050.5,
           Visu_Adv                 := DB51.DBW  628,
           Visu_Ret                 := DB51.DBW  630);
      NOP   0;
NETWORK
TITLE =

      A     M      3.3;
      =     L      0.0;
      BLD   103;
      A(    ;
      O     I     49.6;
      ON    I     49.7;
      )     ;
      =     L      0.1;
      BLD   103;
      A     I     49.7;
      =     L      0.2;
      BLD   103;
      A     Q     57.2;
      =     L      1.1;
      BLD   103;
      A     Q     57.3;
      =     L      1.2;
      BLD   103;
      AN    M   2004.0;
      AN    M   2004.1;
      AN    M   6560.0;
      AN    M   6580.0;
      AN    M   6060.3;
      AN    M   2004.2;
      A     M   2000.2;
      =     L      1.3;
      BLD   103;
      A(    ;
      O     I     80.1;
      O     M   4120.1;
      )     ;
      =     L      1.5;
      BLD   103;
      A     M      0.5;
      =     L      1.6;
      BLD   103;
      CALL #S708_ELE_UP_DN (
           Enable_Aux               := L      0.0,
           Adv_Amount               := 1,
           Ret_Amount               := 1,
           LS_Adv1                  := L      0.1,
           LS_Ret1                  := L      0.2,
           SOL_Adv                  := L      1.1,
           SOL_Ret                  := L      1.2,
           M_Ready                  := L      1.3,
           T_CHK1                   := T#4S,
           T_CHK2                   := T#4S,
           PB_Error_Rst             := L      1.5,
           M_FLICK                  := L      1.6,
           M_Adv_Err                := M   2050.6,
           M_Ret_Err                := M   2050.7,
           Visu_Adv                 := DB51.DBW  636,
           Visu_Ret                 := DB51.DBW  638);
      NOP   0;
NETWORK
TITLE =
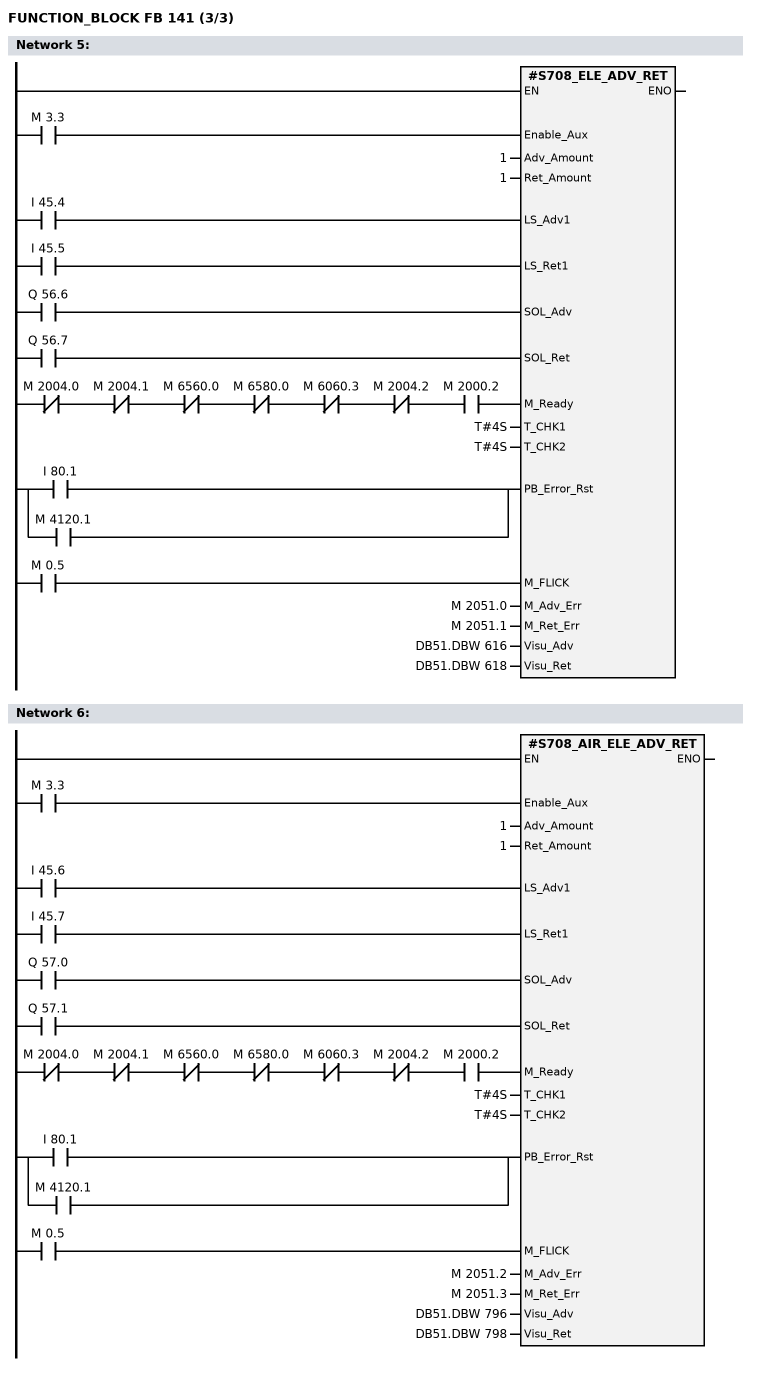

      A     M      3.3;
      =     L      0.0;
      BLD   103;
      A     I     45.4;
      =     L      0.1;
      BLD   103;
      A     I     45.5;
      =     L      0.2;
      BLD   103;
      A     Q     56.6;
      =     L      1.1;
      BLD   103;
      A     Q     56.7;
      =     L      1.2;
      BLD   103;
      AN    M   2004.0;
      AN    M   2004.1;
      AN    M   6560.0;
      AN    M   6580.0;
      AN    M   6060.3;
      AN    M   2004.2;
      A     M   2000.2;
      =     L      1.3;
      BLD   103;
      A(    ;
      O     I     80.1;
      O     M   4120.1;
      )     ;
      =     L      1.5;
      BLD   103;
      A     M      0.5;
      =     L      1.6;
      BLD   103;
      CALL #S708_ELE_ADV_RET (
           Enable_Aux               := L      0.0,
           Adv_Amount               := 1,
           Ret_Amount               := 1,
           LS_Adv1                  := L      0.1,
           LS_Ret1                  := L      0.2,
           SOL_Adv                  := L      1.1,
           SOL_Ret                  := L      1.2,
           M_Ready                  := L      1.3,
           T_CHK1                   := T#4S,
           T_CHK2                   := T#4S,
           PB_Error_Rst             := L      1.5,
           M_FLICK                  := L      1.6,
           M_Adv_Err                := M   2051.0,
           M_Ret_Err                := M   2051.1,
           Visu_Adv                 := DB51.DBW  616,
           Visu_Ret                 := DB51.DBW  618);
      NOP   0;
NETWORK
TITLE =

      A     M      3.3;
      =     L      0.0;
      BLD   103;
      A     I     45.6;
      =     L      0.1;
      BLD   103;
      A     I     45.7;
      =     L      0.2;
      BLD   103;
      A     Q     57.0;
      =     L      1.1;
      BLD   103;
      A     Q     57.1;
      =     L      1.2;
      BLD   103;
      AN    M   2004.0;
      AN    M   2004.1;
      AN    M   6560.0;
      AN    M   6580.0;
      AN    M   6060.3;
      AN    M   2004.2;
      A     M   2000.2;
      =     L      1.3;
      BLD   103;
      A(    ;
      O     I     80.1;
      O     M   4120.1;
      )     ;
      =     L      1.5;
      BLD   103;
      A     M      0.5;
      =     L      1.6;
      BLD   103;
      CALL #S708_AIR_ELE_ADV_RET (
           Enable_Aux               := L      0.0,
           Adv_Amount               := 1,
           Ret_Amount               := 1,
           LS_Adv1                  := L      0.1,
           LS_Ret1                  := L      0.2,
           SOL_Adv                  := L      1.1,
           SOL_Ret                  := L      1.2,
           M_Ready                  := L      1.3,
           T_CHK1                   := T#4S,
           T_CHK2                   := T#4S,
           PB_Error_Rst             := L      1.5,
           M_FLICK                  := L      1.6,
           M_Adv_Err                := M   2051.2,
           M_Ret_Err                := M   2051.3,
           Visu_Adv                 := DB51.DBW  796,
           Visu_Ret                 := DB51.DBW  798);
      NOP   0;
END_FUNCTION_BLOCK

DATA_BLOCK DB 141
TITLE =
VERSION : 0.0

 FB 141
BEGIN
   S708_HOOK_PIN.Enable_Aux := TRUE;
   S708_HOOK_PIN.Adv_Amount := 1;
   S708_HOOK_PIN.Ret_Amount := 1;
   S708_HOOK_PIN.LS_Adv1 := FALSE;
   S708_HOOK_PIN.LS_Ret1 := TRUE;
   S708_HOOK_PIN.LS_Adv2 := FALSE;
   S708_HOOK_PIN.LS_Ret2 := FALSE;
   S708_HOOK_PIN.LS_Adv3 := FALSE;
   S708_HOOK_PIN.LS_Ret3 := FALSE;
   S708_HOOK_PIN.LS_Adv4 := FALSE;
   S708_HOOK_PIN.LS_Ret4 := FALSE;
   S708_HOOK_PIN.SOL_Adv := FALSE;
   S708_HOOK_PIN.SOL_Ret := FALSE;
   S708_HOOK_PIN.M_Ready := TRUE;
   S708_HOOK_PIN.T_CHK1 := T#4S;
   S708_HOOK_PIN.T_CHK2 := T#4S;
   S708_HOOK_PIN.PB_Lamp_CHK := FALSE;
   S708_HOOK_PIN.PB_Error_Rst := FALSE;
   S708_HOOK_PIN.M_FLICK := TRUE;
   S708_HOOK_PIN.M_Adv_Err := FALSE;
   S708_HOOK_PIN.M_Ret_Err := FALSE;
   S708_HOOK_PIN.LP_Adv := FALSE;
   S708_HOOK_PIN.LP_Ret := TRUE;
   S708_HOOK_PIN.Visu_Adv := W#16#0;
   S708_HOOK_PIN.Visu_Ret := W#16#300;
   S708_HOOK_PIN.Error_T1.IN := FALSE;
   S708_HOOK_PIN.Error_T1.PT := T#4S;
   S708_HOOK_PIN.Error_T1.Q := FALSE;
   S708_HOOK_PIN.Error_T1.ET := T#0MS;
   S708_HOOK_PIN.Error_T1.STATE := B#16#0;
   S708_HOOK_PIN.Error_T1.STIME := T#23D5H8M44S147MS;
   S708_HOOK_PIN.Error_T1.ATIME := T#23D5H8M44S516MS;
   S708_HOOK_PIN.Error_T2.IN := FALSE;
   S708_HOOK_PIN.Error_T2.PT := T#4S;
   S708_HOOK_PIN.Error_T2.Q := FALSE;
   S708_HOOK_PIN.Error_T2.ET := T#0MS;
   S708_HOOK_PIN.Error_T2.STATE := B#16#0;
   S708_HOOK_PIN.Error_T2.STIME := T#0MS;
   S708_HOOK_PIN.Error_T2.ATIME := T#0MS;
   S708_HOOK_PIN.CHK_Aux1 := FALSE;
   S708_HOOK_PIN.CHK_Aux2 := FALSE;
   S708_HOOK_PIN.Error_T1_DN := FALSE;
   S708_HOOK_PIN.Error_T2_DN := FALSE;
   S708_HOOK_PIN.Adv_Memo := FALSE;
   S708_HOOK_PIN.Visu_Adv_Arr[0] := FALSE;
   S708_HOOK_PIN.Visu_Adv_Arr[1] := FALSE;
   S708_HOOK_PIN.Visu_Adv_Arr[2] := FALSE;
   S708_HOOK_PIN.Visu_Adv_Arr[3] := FALSE;
   S708_HOOK_PIN.Visu_Adv_Arr[4] := FALSE;
   S708_HOOK_PIN.Visu_Adv_Arr[5] := FALSE;
   S708_HOOK_PIN.Visu_Adv_Arr[6] := FALSE;
   S708_HOOK_PIN.Visu_Adv_Arr[7] := FALSE;
   S708_HOOK_PIN.Visu_Adv_Arr[8] := FALSE;
   S708_HOOK_PIN.Visu_Adv_Arr[9] := FALSE;
   S708_HOOK_PIN.Visu_Adv_Arr[10] := FALSE;
   S708_HOOK_PIN.Visu_Adv_Arr[11] := FALSE;
   S708_HOOK_PIN.Visu_Adv_Arr[12] := FALSE;
   S708_HOOK_PIN.Visu_Adv_Arr[13] := FALSE;
   S708_HOOK_PIN.Visu_Adv_Arr[14] := FALSE;
   S708_HOOK_PIN.Visu_Adv_Arr[15] := FALSE;
   S708_HOOK_PIN.Visu_Ret_Arr[0] := TRUE;
   S708_HOOK_PIN.Visu_Ret_Arr[1] := TRUE;
   S708_HOOK_PIN.Visu_Ret_Arr[2] := FALSE;
   S708_HOOK_PIN.Visu_Ret_Arr[3] := FALSE;
   S708_HOOK_PIN.Visu_Ret_Arr[4] := FALSE;
   S708_HOOK_PIN.Visu_Ret_Arr[5] := FALSE;
   S708_HOOK_PIN.Visu_Ret_Arr[6] := FALSE;
   S708_HOOK_PIN.Visu_Ret_Arr[7] := FALSE;
   S708_HOOK_PIN.Visu_Ret_Arr[8] := FALSE;
   S708_HOOK_PIN.Visu_Ret_Arr[9] := FALSE;
   S708_HOOK_PIN.Visu_Ret_Arr[10] := FALSE;
   S708_HOOK_PIN.Visu_Ret_Arr[11] := FALSE;
   S708_HOOK_PIN.Visu_Ret_Arr[12] := FALSE;
   S708_HOOK_PIN.Visu_Ret_Arr[13] := FALSE;
   S708_HOOK_PIN.Visu_Ret_Arr[14] := FALSE;
   S708_HOOK_PIN.Visu_Ret_Arr[15] := FALSE;
   S708_HOOK_PIN.BLK_Move_Ret := 0;
   S708_HOOK_PIN.Enable := TRUE;
   S708_HOOK_PIN.Adv_End := FALSE;
   S708_HOOK_PIN.Ret_End := TRUE;
   S708_EJECT.Enable_Aux := TRUE;
   S708_EJECT.Adv_Amount := 1;
   S708_EJECT.Ret_Amount := 1;
   S708_EJECT.LS_Adv1 := TRUE;
   S708_EJECT.LS_Ret1 := FALSE;
   S708_EJECT.LS_Adv2 := FALSE;
   S708_EJECT.LS_Ret2 := FALSE;
   S708_EJECT.LS_Adv3 := FALSE;
   S708_EJECT.LS_Ret3 := FALSE;
   S708_EJECT.LS_Adv4 := FALSE;
   S708_EJECT.LS_Ret4 := FALSE;
   S708_EJECT.SOL_Adv := FALSE;
   S708_EJECT.SOL_Ret := FALSE;
   S708_EJECT.M_Ready := TRUE;
   S708_EJECT.T_CHK1 := T#4S;
   S708_EJECT.T_CHK2 := T#4S;
   S708_EJECT.PB_Lamp_CHK := FALSE;
   S708_EJECT.PB_Error_Rst := FALSE;
   S708_EJECT.M_FLICK := TRUE;
   S708_EJECT.M_Adv_Err := FALSE;
   S708_EJECT.M_Ret_Err := FALSE;
   S708_EJECT.LP_Adv := TRUE;
   S708_EJECT.LP_Ret := FALSE;
   S708_EJECT.Visu_Adv := W#16#300;
   S708_EJECT.Visu_Ret := W#16#0;
   S708_EJECT.Error_T1.IN := FALSE;
   S708_EJECT.Error_T1.PT := T#4S;
   S708_EJECT.Error_T1.Q := FALSE;
   S708_EJECT.Error_T1.ET := T#0MS;
   S708_EJECT.Error_T1.STATE := B#16#0;
   S708_EJECT.Error_T1.STIME := T#23D5H9M962MS;
   S708_EJECT.Error_T1.ATIME := T#23D5H9M2S631MS;
   S708_EJECT.Error_T2.IN := FALSE;
   S708_EJECT.Error_T2.PT := T#4S;
   S708_EJECT.Error_T2.Q := FALSE;
   S708_EJECT.Error_T2.ET := T#0MS;
   S708_EJECT.Error_T2.STATE := B#16#0;
   S708_EJECT.Error_T2.STIME := T#0MS;
   S708_EJECT.Error_T2.ATIME := T#0MS;
   S708_EJECT.CHK_Aux1 := FALSE;
   S708_EJECT.CHK_Aux2 := FALSE;
   S708_EJECT.Error_T1_DN := FALSE;
   S708_EJECT.Error_T2_DN := FALSE;
   S708_EJECT.Adv_Memo := TRUE;
   S708_EJECT.Visu_Adv_Arr[0] := TRUE;
   S708_EJECT.Visu_Adv_Arr[1] := TRUE;
   S708_EJECT.Visu_Adv_Arr[2] := FALSE;
   S708_EJECT.Visu_Adv_Arr[3] := FALSE;
   S708_EJECT.Visu_Adv_Arr[4] := FALSE;
   S708_EJECT.Visu_Adv_Arr[5] := FALSE;
   S708_EJECT.Visu_Adv_Arr[6] := FALSE;
   S708_EJECT.Visu_Adv_Arr[7] := FALSE;
   S708_EJECT.Visu_Adv_Arr[8] := FALSE;
   S708_EJECT.Visu_Adv_Arr[9] := FALSE;
   S708_EJECT.Visu_Adv_Arr[10] := FALSE;
   S708_EJECT.Visu_Adv_Arr[11] := FALSE;
   S708_EJECT.Visu_Adv_Arr[12] := FALSE;
   S708_EJECT.Visu_Adv_Arr[13] := FALSE;
   S708_EJECT.Visu_Adv_Arr[14] := FALSE;
   S708_EJECT.Visu_Adv_Arr[15] := FALSE;
   S708_EJECT.Visu_Ret_Arr[0] := FALSE;
   S708_EJECT.Visu_Ret_Arr[1] := FALSE;
   S708_EJECT.Visu_Ret_Arr[2] := FALSE;
   S708_EJECT.Visu_Ret_Arr[3] := FALSE;
   S708_EJECT.Visu_Ret_Arr[4] := FALSE;
   S708_EJECT.Visu_Ret_Arr[5] := FALSE;
   S708_EJECT.Visu_Ret_Arr[6] := FALSE;
   S708_EJECT.Visu_Ret_Arr[7] := FALSE;
   S708_EJECT.Visu_Ret_Arr[8] := FALSE;
   S708_EJECT.Visu_Ret_Arr[9] := FALSE;
   S708_EJECT.Visu_Ret_Arr[10] := FALSE;
   S708_EJECT.Visu_Ret_Arr[11] := FALSE;
   S708_EJECT.Visu_Ret_Arr[12] := FALSE;
   S708_EJECT.Visu_Ret_Arr[13] := FALSE;
   S708_EJECT.Visu_Ret_Arr[14] := FALSE;
   S708_EJECT.Visu_Ret_Arr[15] := FALSE;
   S708_EJECT.BLK_Move_Ret := 0;
   S708_EJECT.Enable := TRUE;
   S708_EJECT.Adv_End := TRUE;
   S708_EJECT.Ret_End := FALSE;
   S708_SAFETY_PIN.Enable_Aux := TRUE;
   S708_SAFETY_PIN.Adv_Amount := 1;
   S708_SAFETY_PIN.Ret_Amount := 1;
   S708_SAFETY_PIN.LS_Adv1 := TRUE;
   S708_SAFETY_PIN.LS_Ret1 := FALSE;
   S708_SAFETY_PIN.LS_Adv2 := FALSE;
   S708_SAFETY_PIN.LS_Ret2 := FALSE;
   S708_SAFETY_PIN.LS_Adv3 := FALSE;
   S708_SAFETY_PIN.LS_Ret3 := FALSE;
   S708_SAFETY_PIN.LS_Adv4 := FALSE;
   S708_SAFETY_PIN.LS_Ret4 := FALSE;
   S708_SAFETY_PIN.SOL_Adv := FALSE;
   S708_SAFETY_PIN.SOL_Ret := FALSE;
   S708_SAFETY_PIN.M_Ready := TRUE;
   S708_SAFETY_PIN.T_CHK1 := T#4S;
   S708_SAFETY_PIN.T_CHK2 := T#4S;
   S708_SAFETY_PIN.PB_Lamp_CHK := FALSE;
   S708_SAFETY_PIN.PB_Error_Rst := FALSE;
   S708_SAFETY_PIN.M_FLICK := TRUE;
   S708_SAFETY_PIN.M_Adv_Err := FALSE;
   S708_SAFETY_PIN.M_Ret_Err := FALSE;
   S708_SAFETY_PIN.LP_Adv := TRUE;
   S708_SAFETY_PIN.LP_Ret := FALSE;
   S708_SAFETY_PIN.Visu_Adv := W#16#300;
   S708_SAFETY_PIN.Visu_Ret := W#16#0;
   S708_SAFETY_PIN.Error_T1.IN := FALSE;
   S708_SAFETY_PIN.Error_T1.PT := T#4S;
   S708_SAFETY_PIN.Error_T1.Q := FALSE;
   S708_SAFETY_PIN.Error_T1.ET := T#0MS;
   S708_SAFETY_PIN.Error_T1.STATE := B#16#0;
   S708_SAFETY_PIN.Error_T1.STIME := T#23D5H8M43S364MS;
   S708_SAFETY_PIN.Error_T1.ATIME := T#23D5H8M43S824MS;
   S708_SAFETY_PIN.Error_T2.IN := FALSE;
   S708_SAFETY_PIN.Error_T2.PT := T#4S;
   S708_SAFETY_PIN.Error_T2.Q := FALSE;
   S708_SAFETY_PIN.Error_T2.ET := T#0MS;
   S708_SAFETY_PIN.Error_T2.STATE := B#16#0;
   S708_SAFETY_PIN.Error_T2.STIME := T#0MS;
   S708_SAFETY_PIN.Error_T2.ATIME := T#0MS;
   S708_SAFETY_PIN.CHK_Aux1 := FALSE;
   S708_SAFETY_PIN.CHK_Aux2 := FALSE;
   S708_SAFETY_PIN.Error_T1_DN := FALSE;
   S708_SAFETY_PIN.Error_T2_DN := FALSE;
   S708_SAFETY_PIN.Adv_Memo := TRUE;
   S708_SAFETY_PIN.Visu_Adv_Arr[0] := TRUE;
   S708_SAFETY_PIN.Visu_Adv_Arr[1] := TRUE;
   S708_SAFETY_PIN.Visu_Adv_Arr[2] := FALSE;
   S708_SAFETY_PIN.Visu_Adv_Arr[3] := FALSE;
   S708_SAFETY_PIN.Visu_Adv_Arr[4] := FALSE;
   S708_SAFETY_PIN.Visu_Adv_Arr[5] := FALSE;
   S708_SAFETY_PIN.Visu_Adv_Arr[6] := FALSE;
   S708_SAFETY_PIN.Visu_Adv_Arr[7] := FALSE;
   S708_SAFETY_PIN.Visu_Adv_Arr[8] := FALSE;
   S708_SAFETY_PIN.Visu_Adv_Arr[9] := FALSE;
   S708_SAFETY_PIN.Visu_Adv_Arr[10] := FALSE;
   S708_SAFETY_PIN.Visu_Adv_Arr[11] := FALSE;
   S708_SAFETY_PIN.Visu_Adv_Arr[12] := FALSE;
   S708_SAFETY_PIN.Visu_Adv_Arr[13] := FALSE;
   S708_SAFETY_PIN.Visu_Adv_Arr[14] := FALSE;
   S708_SAFETY_PIN.Visu_Adv_Arr[15] := FALSE;
   S708_SAFETY_PIN.Visu_Ret_Arr[0] := FALSE;
   S708_SAFETY_PIN.Visu_Ret_Arr[1] := FALSE;
   S708_SAFETY_PIN.Visu_Ret_Arr[2] := FALSE;
   S708_SAFETY_PIN.Visu_Ret_Arr[3] := FALSE;
   S708_SAFETY_PIN.Visu_Ret_Arr[4] := FALSE;
   S708_SAFETY_PIN.Visu_Ret_Arr[5] := FALSE;
   S708_SAFETY_PIN.Visu_Ret_Arr[6] := FALSE;
   S708_SAFETY_PIN.Visu_Ret_Arr[7] := FALSE;
   S708_SAFETY_PIN.Visu_Ret_Arr[8] := FALSE;
   S708_SAFETY_PIN.Visu_Ret_Arr[9] := FALSE;
   S708_SAFETY_PIN.Visu_Ret_Arr[10] := FALSE;
   S708_SAFETY_PIN.Visu_Ret_Arr[11] := FALSE;
   S708_SAFETY_PIN.Visu_Ret_Arr[12] := FALSE;
   S708_SAFETY_PIN.Visu_Ret_Arr[13] := FALSE;
   S708_SAFETY_PIN.Visu_Ret_Arr[14] := FALSE;
   S708_SAFETY_PIN.Visu_Ret_Arr[15] := FALSE;
   S708_SAFETY_PIN.BLK_Move_Ret := 0;
   S708_SAFETY_PIN.Enable := TRUE;
   S708_SAFETY_PIN.Adv_End := TRUE;
   S708_SAFETY_PIN.Ret_End := FALSE;
   S708_ELE_UP_DN.Enable_Aux := TRUE;
   S708_ELE_UP_DN.Adv_Amount := 1;
   S708_ELE_UP_DN.Ret_Amount := 1;
   S708_ELE_UP_DN.LS_Adv1 := TRUE;
   S708_ELE_UP_DN.LS_Ret1 := FALSE;
   S708_ELE_UP_DN.LS_Adv2 := FALSE;
   S708_ELE_UP_DN.LS_Ret2 := FALSE;
   S708_ELE_UP_DN.LS_Adv3 := FALSE;
   S708_ELE_UP_DN.LS_Ret3 := FALSE;
   S708_ELE_UP_DN.LS_Adv4 := FALSE;
   S708_ELE_UP_DN.LS_Ret4 := FALSE;
   S708_ELE_UP_DN.SOL_Adv := FALSE;
   S708_ELE_UP_DN.SOL_Ret := FALSE;
   S708_ELE_UP_DN.M_Ready := TRUE;
   S708_ELE_UP_DN.T_CHK1 := T#4S;
   S708_ELE_UP_DN.T_CHK2 := T#4S;
   S708_ELE_UP_DN.PB_Lamp_CHK := FALSE;
   S708_ELE_UP_DN.PB_Error_Rst := FALSE;
   S708_ELE_UP_DN.M_FLICK := TRUE;
   S708_ELE_UP_DN.M_Adv_Err := FALSE;
   S708_ELE_UP_DN.M_Ret_Err := FALSE;
   S708_ELE_UP_DN.LP_Adv := TRUE;
   S708_ELE_UP_DN.LP_Ret := FALSE;
   S708_ELE_UP_DN.Visu_Adv := W#16#300;
   S708_ELE_UP_DN.Visu_Ret := W#16#0;
   S708_ELE_UP_DN.Error_T1.IN := FALSE;
   S708_ELE_UP_DN.Error_T1.PT := T#4S;
   S708_ELE_UP_DN.Error_T1.Q := FALSE;
   S708_ELE_UP_DN.Error_T1.ET := T#0MS;
   S708_ELE_UP_DN.Error_T1.STATE := B#16#0;
   S708_ELE_UP_DN.Error_T1.STIME := T#-1D3H42M47S140MS;
   S708_ELE_UP_DN.Error_T1.ATIME := T#-1D3H42M43S131MS;
   S708_ELE_UP_DN.Error_T2.IN := FALSE;
   S708_ELE_UP_DN.Error_T2.PT := T#4S;
   S708_ELE_UP_DN.Error_T2.Q := FALSE;
   S708_ELE_UP_DN.Error_T2.ET := T#0MS;
   S708_ELE_UP_DN.Error_T2.STATE := B#16#0;
   S708_ELE_UP_DN.Error_T2.STIME := T#0MS;
   S708_ELE_UP_DN.Error_T2.ATIME := T#0MS;
   S708_ELE_UP_DN.CHK_Aux1 := FALSE;
   S708_ELE_UP_DN.CHK_Aux2 := FALSE;
   S708_ELE_UP_DN.Error_T1_DN := FALSE;
   S708_ELE_UP_DN.Error_T2_DN := FALSE;
   S708_ELE_UP_DN.Adv_Memo := TRUE;
   S708_ELE_UP_DN.Visu_Adv_Arr[0] := TRUE;
   S708_ELE_UP_DN.Visu_Adv_Arr[1] := TRUE;
   S708_ELE_UP_DN.Visu_Adv_Arr[2] := FALSE;
   S708_ELE_UP_DN.Visu_Adv_Arr[3] := FALSE;
   S708_ELE_UP_DN.Visu_Adv_Arr[4] := FALSE;
   S708_ELE_UP_DN.Visu_Adv_Arr[5] := FALSE;
   S708_ELE_UP_DN.Visu_Adv_Arr[6] := FALSE;
   S708_ELE_UP_DN.Visu_Adv_Arr[7] := FALSE;
   S708_ELE_UP_DN.Visu_Adv_Arr[8] := FALSE;
   S708_ELE_UP_DN.Visu_Adv_Arr[9] := FALSE;
   S708_ELE_UP_DN.Visu_Adv_Arr[10] := FALSE;
   S708_ELE_UP_DN.Visu_Adv_Arr[11] := FALSE;
   S708_ELE_UP_DN.Visu_Adv_Arr[12] := FALSE;
   S708_ELE_UP_DN.Visu_Adv_Arr[13] := FALSE;
   S708_ELE_UP_DN.Visu_Adv_Arr[14] := FALSE;
   S708_ELE_UP_DN.Visu_Adv_Arr[15] := FALSE;
   S708_ELE_UP_DN.Visu_Ret_Arr[0] := FALSE;
   S708_ELE_UP_DN.Visu_Ret_Arr[1] := FALSE;
   S708_ELE_UP_DN.Visu_Ret_Arr[2] := FALSE;
   S708_ELE_UP_DN.Visu_Ret_Arr[3] := FALSE;
   S708_ELE_UP_DN.Visu_Ret_Arr[4] := FALSE;
   S708_ELE_UP_DN.Visu_Ret_Arr[5] := FALSE;
   S708_ELE_UP_DN.Visu_Ret_Arr[6] := FALSE;
   S708_ELE_UP_DN.Visu_Ret_Arr[7] := FALSE;
   S708_ELE_UP_DN.Visu_Ret_Arr[8] := FALSE;
   S708_ELE_UP_DN.Visu_Ret_Arr[9] := FALSE;
   S708_ELE_UP_DN.Visu_Ret_Arr[10] := FALSE;
   S708_ELE_UP_DN.Visu_Ret_Arr[11] := FALSE;
   S708_ELE_UP_DN.Visu_Ret_Arr[12] := FALSE;
   S708_ELE_UP_DN.Visu_Ret_Arr[13] := FALSE;
   S708_ELE_UP_DN.Visu_Ret_Arr[14] := FALSE;
   S708_ELE_UP_DN.Visu_Ret_Arr[15] := FALSE;
   S708_ELE_UP_DN.BLK_Move_Ret := 0;
   S708_ELE_UP_DN.Enable := TRUE;
   S708_ELE_UP_DN.Adv_End := TRUE;
   S708_ELE_UP_DN.Ret_End := FALSE;
   S708_ELE_ADV_RET.Enable_Aux := TRUE;
   S708_ELE_ADV_RET.Adv_Amount := 1;
   S708_ELE_ADV_RET.Ret_Amount := 1;
   S708_ELE_ADV_RET.LS_Adv1 := FALSE;
   S708_ELE_ADV_RET.LS_Ret1 := TRUE;
   S708_ELE_ADV_RET.LS_Adv2 := FALSE;
   S708_ELE_ADV_RET.LS_Ret2 := FALSE;
   S708_ELE_ADV_RET.LS_Adv3 := FALSE;
   S708_ELE_ADV_RET.LS_Ret3 := FALSE;
   S708_ELE_ADV_RET.LS_Adv4 := FALSE;
   S708_ELE_ADV_RET.LS_Ret4 := FALSE;
   S708_ELE_ADV_RET.SOL_Adv := FALSE;
   S708_ELE_ADV_RET.SOL_Ret := FALSE;
   S708_ELE_ADV_RET.M_Ready := TRUE;
   S708_ELE_ADV_RET.T_CHK1 := T#4S;
   S708_ELE_ADV_RET.T_CHK2 := T#4S;
   S708_ELE_ADV_RET.PB_Lamp_CHK := FALSE;
   S708_ELE_ADV_RET.PB_Error_Rst := FALSE;
   S708_ELE_ADV_RET.M_FLICK := TRUE;
   S708_ELE_ADV_RET.M_Adv_Err := FALSE;
   S708_ELE_ADV_RET.M_Ret_Err := FALSE;
   S708_ELE_ADV_RET.LP_Adv := FALSE;
   S708_ELE_ADV_RET.LP_Ret := TRUE;
   S708_ELE_ADV_RET.Visu_Adv := W#16#0;
   S708_ELE_ADV_RET.Visu_Ret := W#16#300;
   S708_ELE_ADV_RET.Error_T1.IN := FALSE;
   S708_ELE_ADV_RET.Error_T1.PT := T#4S;
   S708_ELE_ADV_RET.Error_T1.Q := FALSE;
   S708_ELE_ADV_RET.Error_T1.ET := T#0MS;
   S708_ELE_ADV_RET.Error_T1.STATE := B#16#0;
   S708_ELE_ADV_RET.Error_T1.STIME := T#23D5H9M804MS;
   S708_ELE_ADV_RET.Error_T1.ATIME := T#23D5H9M939MS;
   S708_ELE_ADV_RET.Error_T2.IN := FALSE;
   S708_ELE_ADV_RET.Error_T2.PT := T#4S;
   S708_ELE_ADV_RET.Error_T2.Q := FALSE;
   S708_ELE_ADV_RET.Error_T2.ET := T#0MS;
   S708_ELE_ADV_RET.Error_T2.STATE := B#16#0;
   S708_ELE_ADV_RET.Error_T2.STIME := T#0MS;
   S708_ELE_ADV_RET.Error_T2.ATIME := T#0MS;
   S708_ELE_ADV_RET.CHK_Aux1 := FALSE;
   S708_ELE_ADV_RET.CHK_Aux2 := FALSE;
   S708_ELE_ADV_RET.Error_T1_DN := FALSE;
   S708_ELE_ADV_RET.Error_T2_DN := FALSE;
   S708_ELE_ADV_RET.Adv_Memo := FALSE;
   S708_ELE_ADV_RET.Visu_Adv_Arr[0] := FALSE;
   S708_ELE_ADV_RET.Visu_Adv_Arr[1] := FALSE;
   S708_ELE_ADV_RET.Visu_Adv_Arr[2] := FALSE;
   S708_ELE_ADV_RET.Visu_Adv_Arr[3] := FALSE;
   S708_ELE_ADV_RET.Visu_Adv_Arr[4] := FALSE;
   S708_ELE_ADV_RET.Visu_Adv_Arr[5] := FALSE;
   S708_ELE_ADV_RET.Visu_Adv_Arr[6] := FALSE;
   S708_ELE_ADV_RET.Visu_Adv_Arr[7] := FALSE;
   S708_ELE_ADV_RET.Visu_Adv_Arr[8] := FALSE;
   S708_ELE_ADV_RET.Visu_Adv_Arr[9] := FALSE;
   S708_ELE_ADV_RET.Visu_Adv_Arr[10] := FALSE;
   S708_ELE_ADV_RET.Visu_Adv_Arr[11] := FALSE;
   S708_ELE_ADV_RET.Visu_Adv_Arr[12] := FALSE;
   S708_ELE_ADV_RET.Visu_Adv_Arr[13] := FALSE;
   S708_ELE_ADV_RET.Visu_Adv_Arr[14] := FALSE;
   S708_ELE_ADV_RET.Visu_Adv_Arr[15] := FALSE;
   S708_ELE_ADV_RET.Visu_Ret_Arr[0] := TRUE;
   S708_ELE_ADV_RET.Visu_Ret_Arr[1] := TRUE;
   S708_ELE_ADV_RET.Visu_Ret_Arr[2] := FALSE;
   S708_ELE_ADV_RET.Visu_Ret_Arr[3] := FALSE;
   S708_ELE_ADV_RET.Visu_Ret_Arr[4] := FALSE;
   S708_ELE_ADV_RET.Visu_Ret_Arr[5] := FALSE;
   S708_ELE_ADV_RET.Visu_Ret_Arr[6] := FALSE;
   S708_ELE_ADV_RET.Visu_Ret_Arr[7] := FALSE;
   S708_ELE_ADV_RET.Visu_Ret_Arr[8] := FALSE;
   S708_ELE_ADV_RET.Visu_Ret_Arr[9] := FALSE;
   S708_ELE_ADV_RET.Visu_Ret_Arr[10] := FALSE;
   S708_ELE_ADV_RET.Visu_Ret_Arr[11] := FALSE;
   S708_ELE_ADV_RET.Visu_Ret_Arr[12] := FALSE;
   S708_ELE_ADV_RET.Visu_Ret_Arr[13] := FALSE;
   S708_ELE_ADV_RET.Visu_Ret_Arr[14] := FALSE;
   S708_ELE_ADV_RET.Visu_Ret_Arr[15] := FALSE;
   S708_ELE_ADV_RET.BLK_Move_Ret := 0;
   S708_ELE_ADV_RET.Enable := TRUE;
   S708_ELE_ADV_RET.Adv_End := FALSE;
   S708_ELE_ADV_RET.Ret_End := TRUE;
   S708_AIR_ELE_ADV_RET.Enable_Aux := TRUE;
   S708_AIR_ELE_ADV_RET.Adv_Amount := 1;
   S708_AIR_ELE_ADV_RET.Ret_Amount := 1;
   S708_AIR_ELE_ADV_RET.LS_Adv1 := FALSE;
   S708_AIR_ELE_ADV_RET.LS_Ret1 := TRUE;
   S708_AIR_ELE_ADV_RET.LS_Adv2 := FALSE;
   S708_AIR_ELE_ADV_RET.LS_Ret2 := FALSE;
   S708_AIR_ELE_ADV_RET.LS_Adv3 := FALSE;
   S708_AIR_ELE_ADV_RET.LS_Ret3 := FALSE;
   S708_AIR_ELE_ADV_RET.LS_Adv4 := FALSE;
   S708_AIR_ELE_ADV_RET.LS_Ret4 := FALSE;
   S708_AIR_ELE_ADV_RET.SOL_Adv := FALSE;
   S708_AIR_ELE_ADV_RET.SOL_Ret := FALSE;
   S708_AIR_ELE_ADV_RET.M_Ready := TRUE;
   S708_AIR_ELE_ADV_RET.T_CHK1 := T#4S;
   S708_AIR_ELE_ADV_RET.T_CHK2 := T#4S;
   S708_AIR_ELE_ADV_RET.PB_Lamp_CHK := FALSE;
   S708_AIR_ELE_ADV_RET.PB_Error_Rst := FALSE;
   S708_AIR_ELE_ADV_RET.M_FLICK := TRUE;
   S708_AIR_ELE_ADV_RET.M_Adv_Err := FALSE;
   S708_AIR_ELE_ADV_RET.M_Ret_Err := FALSE;
   S708_AIR_ELE_ADV_RET.LP_Adv := FALSE;
   S708_AIR_ELE_ADV_RET.LP_Ret := TRUE;
   S708_AIR_ELE_ADV_RET.Visu_Adv := W#16#0;
   S708_AIR_ELE_ADV_RET.Visu_Ret := W#16#300;
   S708_AIR_ELE_ADV_RET.Error_T1.IN := FALSE;
   S708_AIR_ELE_ADV_RET.Error_T1.PT := T#4S;
   S708_AIR_ELE_ADV_RET.Error_T1.Q := FALSE;
   S708_AIR_ELE_ADV_RET.Error_T1.ET := T#0MS;
   S708_AIR_ELE_ADV_RET.Error_T1.STATE := B#16#0;
   S708_AIR_ELE_ADV_RET.Error_T1.STIME := T#23D5H9M300MS;
   S708_AIR_ELE_ADV_RET.Error_T1.ATIME := T#23D5H9M485MS;
   S708_AIR_ELE_ADV_RET.Error_T2.IN := FALSE;
   S708_AIR_ELE_ADV_RET.Error_T2.PT := T#4S;
   S708_AIR_ELE_ADV_RET.Error_T2.Q := FALSE;
   S708_AIR_ELE_ADV_RET.Error_T2.ET := T#0MS;
   S708_AIR_ELE_ADV_RET.Error_T2.STATE := B#16#0;
   S708_AIR_ELE_ADV_RET.Error_T2.STIME := T#0MS;
   S708_AIR_ELE_ADV_RET.Error_T2.ATIME := T#0MS;
   S708_AIR_ELE_ADV_RET.CHK_Aux1 := FALSE;
   S708_AIR_ELE_ADV_RET.CHK_Aux2 := FALSE;
   S708_AIR_ELE_ADV_RET.Error_T1_DN := FALSE;
   S708_AIR_ELE_ADV_RET.Error_T2_DN := FALSE;
   S708_AIR_ELE_ADV_RET.Adv_Memo := FALSE;
   S708_AIR_ELE_ADV_RET.Visu_Adv_Arr[0] := FALSE;
   S708_AIR_ELE_ADV_RET.Visu_Adv_Arr[1] := FALSE;
   S708_AIR_ELE_ADV_RET.Visu_Adv_Arr[2] := FALSE;
   S708_AIR_ELE_ADV_RET.Visu_Adv_Arr[3] := FALSE;
   S708_AIR_ELE_ADV_RET.Visu_Adv_Arr[4] := FALSE;
   S708_AIR_ELE_ADV_RET.Visu_Adv_Arr[5] := FALSE;
   S708_AIR_ELE_ADV_RET.Visu_Adv_Arr[6] := FALSE;
   S708_AIR_ELE_ADV_RET.Visu_Adv_Arr[7] := FALSE;
   S708_AIR_ELE_ADV_RET.Visu_Adv_Arr[8] := FALSE;
   S708_AIR_ELE_ADV_RET.Visu_Adv_Arr[9] := FALSE;
   S708_AIR_ELE_ADV_RET.Visu_Adv_Arr[10] := FALSE;
   S708_AIR_ELE_ADV_RET.Visu_Adv_Arr[11] := FALSE;
   S708_AIR_ELE_ADV_RET.Visu_Adv_Arr[12] := FALSE;
   S708_AIR_ELE_ADV_RET.Visu_Adv_Arr[13] := FALSE;
   S708_AIR_ELE_ADV_RET.Visu_Adv_Arr[14] := FALSE;
   S708_AIR_ELE_ADV_RET.Visu_Adv_Arr[15] := FALSE;
   S708_AIR_ELE_ADV_RET.Visu_Ret_Arr[0] := TRUE;
   S708_AIR_ELE_ADV_RET.Visu_Ret_Arr[1] := TRUE;
   S708_AIR_ELE_ADV_RET.Visu_Ret_Arr[2] := FALSE;
   S708_AIR_ELE_ADV_RET.Visu_Ret_Arr[3] := FALSE;
   S708_AIR_ELE_ADV_RET.Visu_Ret_Arr[4] := FALSE;
   S708_AIR_ELE_ADV_RET.Visu_Ret_Arr[5] := FALSE;
   S708_AIR_ELE_ADV_RET.Visu_Ret_Arr[6] := FALSE;
   S708_AIR_ELE_ADV_RET.Visu_Ret_Arr[7] := FALSE;
   S708_AIR_ELE_ADV_RET.Visu_Ret_Arr[8] := FALSE;
   S708_AIR_ELE_ADV_RET.Visu_Ret_Arr[9] := FALSE;
   S708_AIR_ELE_ADV_RET.Visu_Ret_Arr[10] := FALSE;
   S708_AIR_ELE_ADV_RET.Visu_Ret_Arr[11] := FALSE;
   S708_AIR_ELE_ADV_RET.Visu_Ret_Arr[12] := FALSE;
   S708_AIR_ELE_ADV_RET.Visu_Ret_Arr[13] := FALSE;
   S708_AIR_ELE_ADV_RET.Visu_Ret_Arr[14] := FALSE;
   S708_AIR_ELE_ADV_RET.Visu_Ret_Arr[15] := FALSE;
   S708_AIR_ELE_ADV_RET.BLK_Move_Ret := 0;
   S708_AIR_ELE_ADV_RET.Enable := TRUE;
   S708_AIR_ELE_ADV_RET.Adv_End := FALSE;
   S708_AIR_ELE_ADV_RET.Ret_End := TRUE;
END_DATA_BLOCK

FUNCTION FC 141 : VOID
TITLE =
VERSION : 0.1

BEGIN
NETWORK
TITLE =
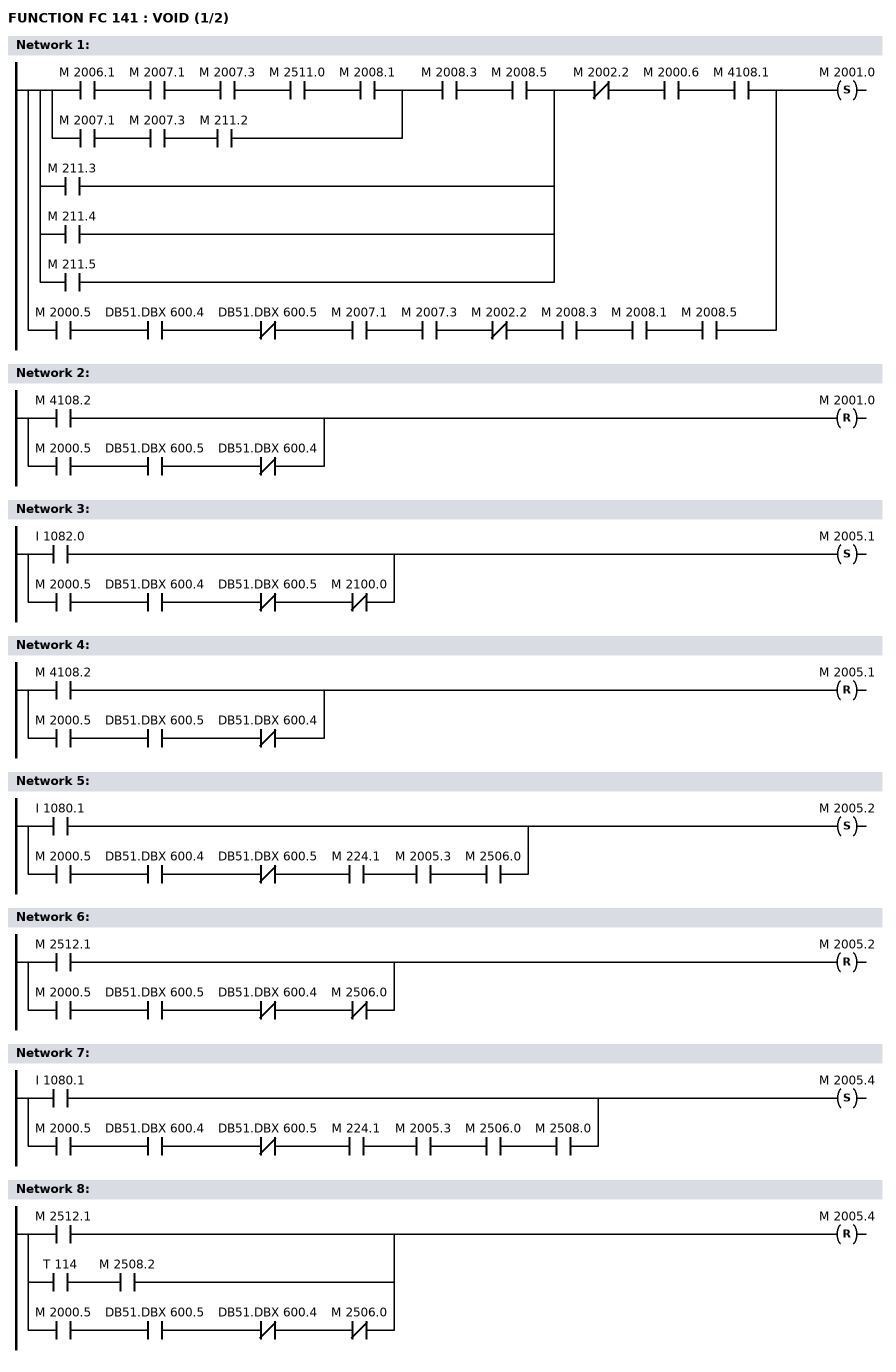

      A(    ;
      A(    ;
      A     M   2006.1;
      A     M   2007.1;
      A     M   2007.3;
      A     M   2511.0;
      A     M   2008.1;
      O     ;
      A     M   2007.1;
      A     M   2007.3;
      A     M    211.2;
      )     ;
      A     M   2008.3;
      A     M   2008.5;
      O     M    211.3;
      O     M    211.4;
      O     M    211.5;
      )     ;
      AN    M   2002.2;
      A     M   2000.6;
      A     M   4108.1;
      O     ;
      A     M   2000.5;
      A     DB51.DBX  600.4;
      AN    DB51.DBX  600.5;
      A     M   2007.1;
      A     M   2007.3;
      AN    M   2002.2;
      A     M   2008.3;
      A     M   2008.1;
      A     M   2008.5;
      S     M   2001.0;
NETWORK
TITLE =

      O     M   4108.2;
      O     ;
      A     M   2000.5;
      A     DB51.DBX  600.5;
      AN    DB51.DBX  600.4;
      R     M   2001.0;
NETWORK
TITLE =

      O     I   1082.0;
      O     ;
      A     M   2000.5;
      A     DB51.DBX  600.4;
      AN    DB51.DBX  600.5;
      AN    M   2100.0;
      S     M   2005.1;
NETWORK
TITLE =

      O     M   4108.2;
      O     ;
      A     M   2000.5;
      A     DB51.DBX  600.5;
      AN    DB51.DBX  600.4;
      R     M   2005.1;
NETWORK
TITLE =

      O     I   1080.1;
      O     ;
      A     M   2000.5;
      A     DB51.DBX  600.4;
      AN    DB51.DBX  600.5;
      A     M    224.1;
      A     M   2005.3;
      A     M   2506.0;
      S     M   2005.2;
NETWORK
TITLE =

      O     M   2512.1;
      O     ;
      A     M   2000.5;
      A     DB51.DBX  600.5;
      AN    DB51.DBX  600.4;
      AN    M   2506.0;
      R     M   2005.2;
NETWORK
TITLE =

      O     I   1080.1;
      O     ;
      A     M   2000.5;
      A     DB51.DBX  600.4;
      AN    DB51.DBX  600.5;
      A     M    224.1;
      A     M   2005.3;
      A     M   2506.0;
      A     M   2508.0;
      S     M   2005.4;
NETWORK
TITLE =

      O     M   2512.1;
      O     ;
      A     T    114;
      A     M   2508.2;
      O     ;
      A     M   2000.5;
      A     DB51.DBX  600.5;
      AN    DB51.DBX  600.4;
      AN    M   2506.0;
      R     M   2005.4;
NETWORK
TITLE =
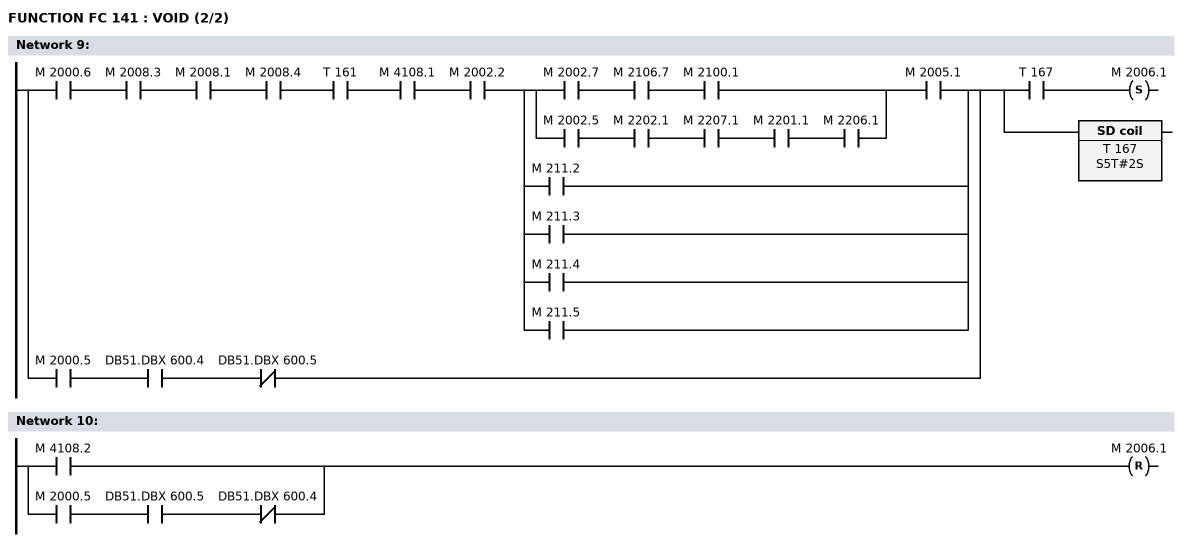

      A     M   2000.6;
      A     M   2008.3;
      A     M   2008.1;
      A     M   2008.4;
      A     T    161;
      A     M   4108.1;
      A     M   2002.2;
      A(    ;
      A(    ;
      A     M   2002.7;
      A     M   2106.7;
      A     M   2100.1;
      O     ;
      A     M   2002.5;
      A     M   2202.1;
      A     M   2207.1;
      A     M   2201.1;
      A     M   2206.1;
      )     ;
      A     M   2005.1;
      O     M    211.2;
      O     M    211.3;
      O     M    211.4;
      O     M    211.5;
      )     ;
      O     ;
      A     M   2000.5;
      A     DB51.DBX  600.4;
      AN    DB51.DBX  600.5;
      =     L      0.0;
      A     L      0.0;
      A     T    167;
      S     M   2006.1;
      A     L      0.0;
      BLD   102;
      L     S5T#2S;
      SD    T    167;
NETWORK
TITLE =

      O     M   4108.2;
      O     ;
      A     M   2000.5;
      A     DB51.DBX  600.5;
      AN    DB51.DBX  600.4;
      R     M   2006.1;
END_FUNCTION

FUNCTION_BLOCK FB 142
TITLE =
VERSION : 0.1

BEGIN
NETWORK
TITLE =
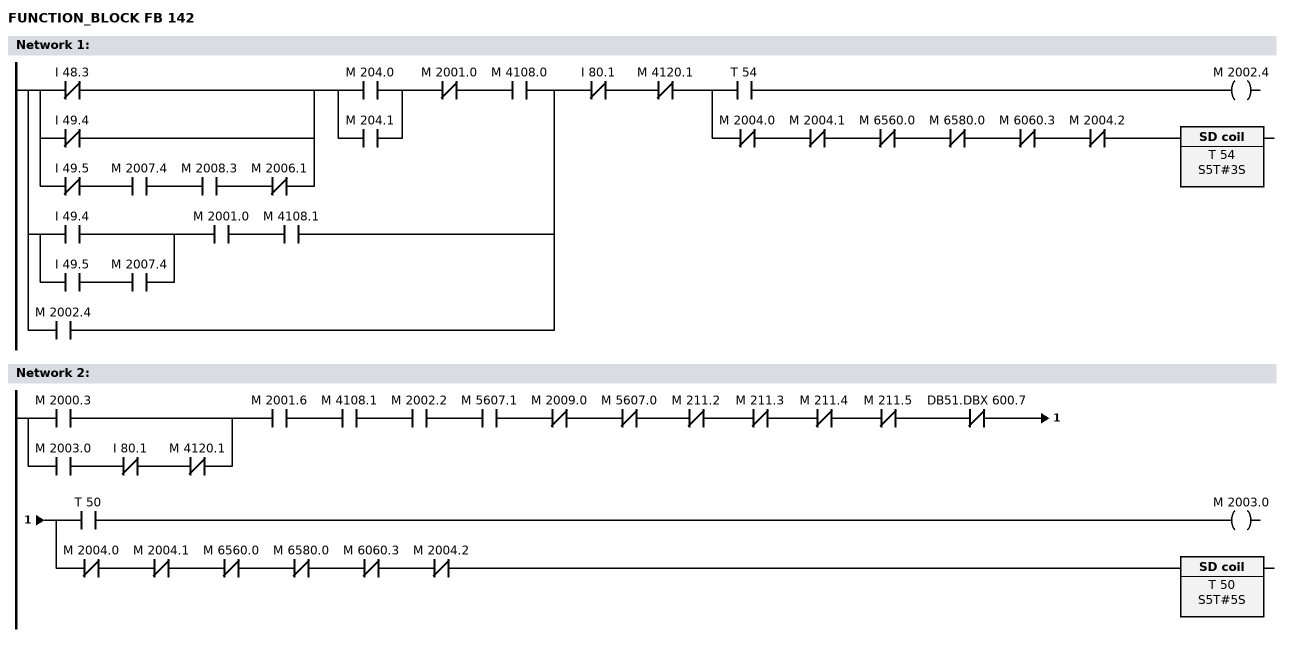

      A(    ;
      A(    ;
      ON    I     48.3;
      ON    I     49.4;
      O     ;
      AN    I     49.5;
      A     M   2007.4;
      A     M   2008.3;
      AN    M   2006.1;
      )     ;
      A(    ;
      O     M    204.0;
      O     M    204.1;
      )     ;
      AN    M   2001.0;
      A     M   4108.0;
      O     ;
      A(    ;
      O     I     49.4;
      O     ;
      A     I     49.5;
      A     M   2007.4;
      )     ;
      A     M   2001.0;
      A     M   4108.1;
      O     M   2002.4;
      )     ;
      AN    I     80.1;
      AN    M   4120.1;
      =     L      0.0;
      A     L      0.0;
      A     T     54;
      =     M   2002.4;
      A     L      0.0;
      AN    M   2004.0;
      AN    M   2004.1;
      AN    M   6560.0;
      AN    M   6580.0;
      AN    M   6060.3;
      AN    M   2004.2;
      L     S5T#3S;
      SD    T     54;
NETWORK
TITLE =

      A(    ;
      O     M   2000.3;
      O     ;
      A     M   2003.0;
      AN    I     80.1;
      AN    M   4120.1;
      )     ;
      A     M   2001.6;
      A     M   4108.1;
      A     M   2002.2;
      A     M   5607.1;
      AN    M   2009.0;
      AN    M   5607.0;
      AN    M    211.2;
      AN    M    211.3;
      AN    M    211.4;
      AN    M    211.5;
      AN    DB51.DBX  600.7;
      =     L      0.0;
      A     L      0.0;
      A     T     50;
      =     M   2003.0;
      A     L      0.0;
      AN    M   2004.0;
      AN    M   2004.1;
      AN    M   6560.0;
      AN    M   6580.0;
      AN    M   6060.3;
      AN    M   2004.2;
      L     S5T#5S;
      SD    T     50;
NETWORK
TITLE =

      A     M   2001.6;
      A     M   2005.1;
      A(    ;
      A     M   2002.7;
      A(    ;
      A     I    268.6;
      A     OV;
      AN    I    268.7;
      O     ;
      AN    I    268.6;
      A     I    268.7;
      O     ;
      A     I    268.6;
      A     I    268.7;
      )     ;
      O     ;
      A     M   2002.5;
      A(    ;
      A     I    370.0;
      A     I    370.1;
      O     ;
      A     I    370.0;
      AN    I    370.1;
      O     ;
      AN    I    370.0;
      A     I    370.1;
      )     ;
      )     ;
      =     L      0.0;
      A     L      0.0;
      A     T     53;
      =     M   2003.1;
      A     L      0.0;
      AN    M   2004.0;
      AN    M   2004.1;
      AN    M   6560.0;
      AN    M   6580.0;
      AN    M   6060.3;
      AN    M   2004.2;
      L     S5T#1S;
      SD    T     53;
NETWORK
TITLE =
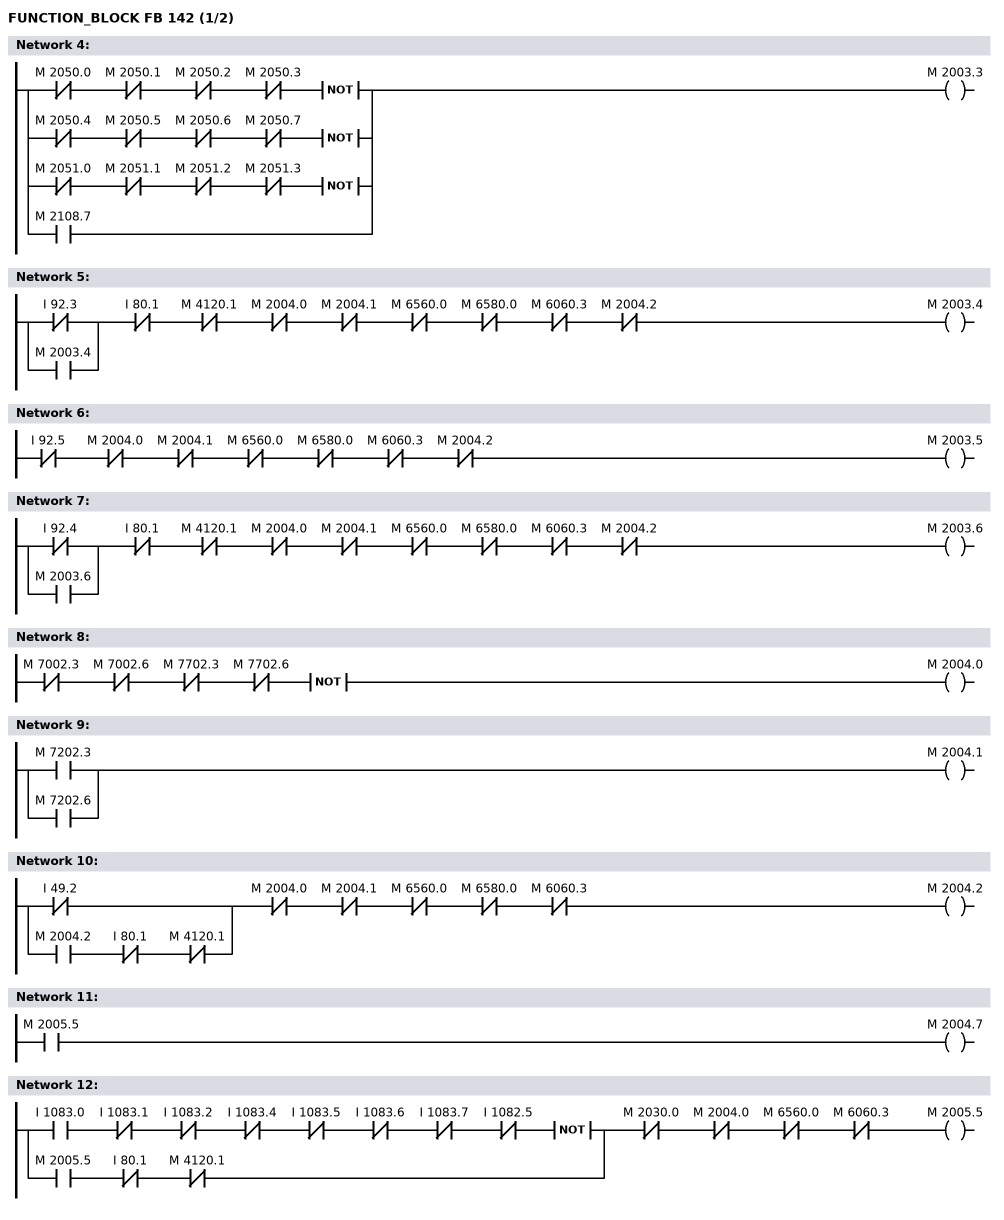

      AN    M   2050.0;
      AN    M   2050.1;
      AN    M   2050.2;
      AN    M   2050.3;
      NOT   ;
      O(    ;
      AN    M   2050.4;
      AN    M   2050.5;
      AN    M   2050.6;
      AN    M   2050.7;
      NOT   ;
      )     ;
      O(    ;
      AN    M   2051.0;
      AN    M   2051.1;
      AN    M   2051.2;
      AN    M   2051.3;
      NOT   ;
      )     ;
      O     M   2108.7;
      =     M   2003.3;
NETWORK
TITLE =

      A(    ;
      ON    I     92.3;
      O     M   2003.4;
      )     ;
      AN    I     80.1;
      AN    M   4120.1;
      AN    M   2004.0;
      AN    M   2004.1;
      AN    M   6560.0;
      AN    M   6580.0;
      AN    M   6060.3;
      AN    M   2004.2;
      =     M   2003.4;
NETWORK
TITLE =

      AN    I     92.5;
      AN    M   2004.0;
      AN    M   2004.1;
      AN    M   6560.0;
      AN    M   6580.0;
      AN    M   6060.3;
      AN    M   2004.2;
      =     M   2003.5;
NETWORK
TITLE =

      A(    ;
      ON    I     92.4;
      O     M   2003.6;
      )     ;
      AN    I     80.1;
      AN    M   4120.1;
      AN    M   2004.0;
      AN    M   2004.1;
      AN    M   6560.0;
      AN    M   6580.0;
      AN    M   6060.3;
      AN    M   2004.2;
      =     M   2003.6;
NETWORK
TITLE =

      AN    M   7002.3;
      AN    M   7002.6;
      AN    M   7702.3;
      AN    M   7702.6;
      NOT   ;
      =     M   2004.0;
NETWORK
TITLE =

      O     M   7202.3;
      O     M   7202.6;
      =     M   2004.1;
NETWORK
TITLE =

      A(    ;
      ON    I     49.2;
      O     ;
      A     M   2004.2;
      AN    I     80.1;
      AN    M   4120.1;
      )     ;
      AN    M   2004.0;
      AN    M   2004.1;
      AN    M   6560.0;
      AN    M   6580.0;
      AN    M   6060.3;
      =     M   2004.2;
NETWORK
TITLE =

      A     M   2005.5;
      =     M   2004.7;
NETWORK
TITLE =

      A(    ;
      A     I   1083.0;
      AN    I   1083.1;
      AN    I   1083.2;
      AN    I   1083.4;
      AN    I   1083.5;
      AN    I   1083.6;
      AN    I   1083.7;
      AN    I   1082.5;
      NOT   ;
      O     ;
      A     M   2005.5;
      AN    I     80.1;
      AN    M   4120.1;
      )     ;
      AN    M   2030.0;
      AN    M   2004.0;
      AN    M   6560.0;
      AN    M   6060.3;
      =     M   2005.5;
NETWORK
TITLE =
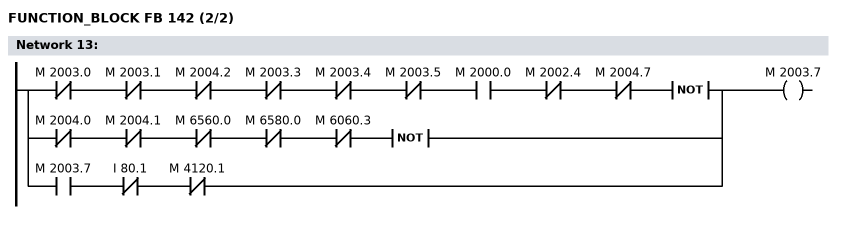

      AN    M   2003.0;
      AN    M   2003.1;
      AN    M   2004.2;
      AN    M   2003.3;
      AN    M   2003.4;
      AN    M   2003.5;
      A     M   2000.0;
      AN    M   2002.4;
      AN    M   2004.7;
      NOT   ;
      O(    ;
      AN    M   2004.0;
      AN    M   2004.1;
      AN    M   6560.0;
      AN    M   6580.0;
      AN    M   6060.3;
      NOT   ;
      )     ;
      O     ;
      A     M   2003.7;
      AN    I     80.1;
      AN    M   4120.1;
      =     M   2003.7;
END_FUNCTION_BLOCK

DATA_BLOCK DB 142
TITLE =
VERSION : 0.0

 FB 142
BEGIN
END_DATA_BLOCK

FUNCTION FC 142 : VOID
TITLE =
VERSION : 0.1

BEGIN
NETWORK
TITLE =
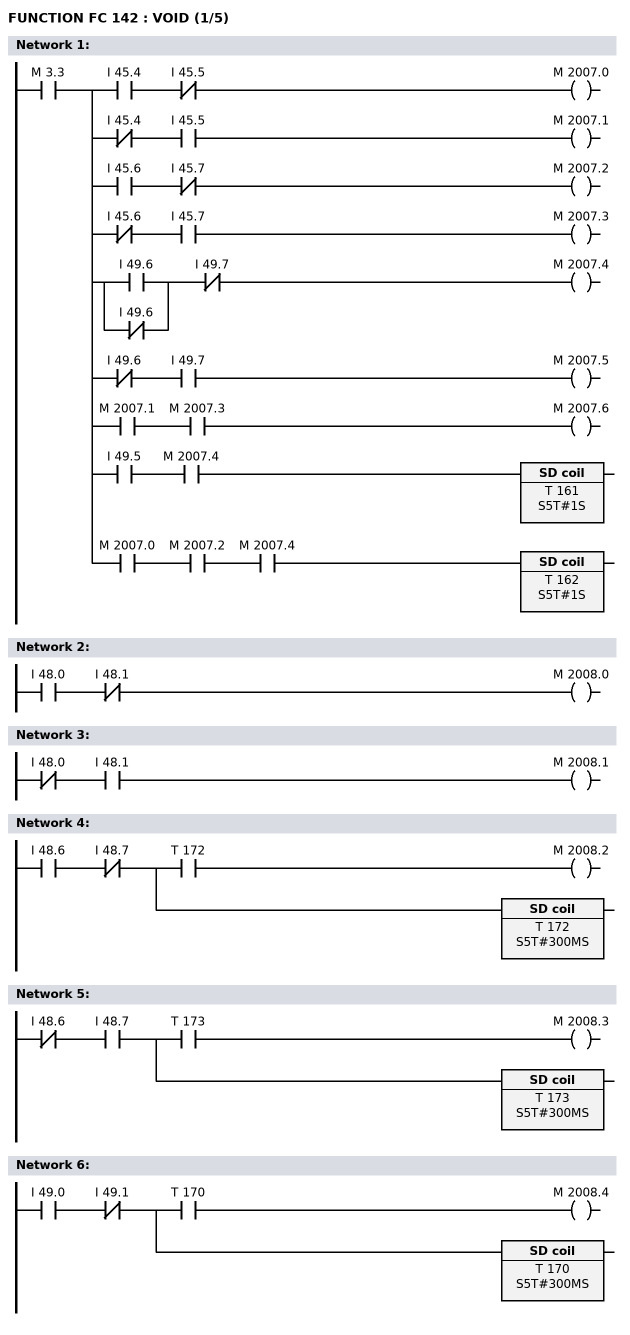

      A     M      3.3;
      =     L      0.0;
      A     L      0.0;
      A     I     45.4;
      AN    I     45.5;
      =     M   2007.0;
      A     L      0.0;
      AN    I     45.4;
      A     I     45.5;
      =     M   2007.1;
      A     L      0.0;
      A     I     45.6;
      AN    I     45.7;
      =     M   2007.2;
      A     L      0.0;
      AN    I     45.6;
      A     I     45.7;
      =     M   2007.3;
      A     L      0.0;
      A(    ;
      O     I     49.6;
      ON    I     49.6;
      )     ;
      AN    I     49.7;
      =     M   2007.4;
      A     L      0.0;
      AN    I     49.6;
      A     I     49.7;
      =     M   2007.5;
      A     L      0.0;
      A     M   2007.1;
      A     M   2007.3;
      =     M   2007.6;
      A     L      0.0;
      A     I     49.5;
      A     M   2007.4;
      L     S5T#1S;
      SD    T    161;
      A     L      0.0;
      A     M   2007.0;
      A     M   2007.2;
      A     M   2007.4;
      L     S5T#1S;
      SD    T    162;
NETWORK
TITLE =

      A     I     48.0;
      AN    I     48.1;
      =     M   2008.0;
NETWORK
TITLE =

      AN    I     48.0;
      A     I     48.1;
      =     M   2008.1;
NETWORK
TITLE =

      A     I     48.6;
      AN    I     48.7;
      =     L      0.0;
      A     L      0.0;
      A     T    172;
      =     M   2008.2;
      A     L      0.0;
      BLD   102;
      L     S5T#300MS;
      SD    T    172;
NETWORK
TITLE =

      AN    I     48.6;
      A     I     48.7;
      =     L      0.0;
      A     L      0.0;
      A     T    173;
      =     M   2008.3;
      A     L      0.0;
      BLD   102;
      L     S5T#300MS;
      SD    T    173;
NETWORK
TITLE =

      A     I     49.0;
      AN    I     49.1;
      =     L      0.0;
      A     L      0.0;
      A     T    170;
      =     M   2008.4;
      A     L      0.0;
      BLD   102;
      L     S5T#300MS;
      SD    T    170;
NETWORK
TITLE =
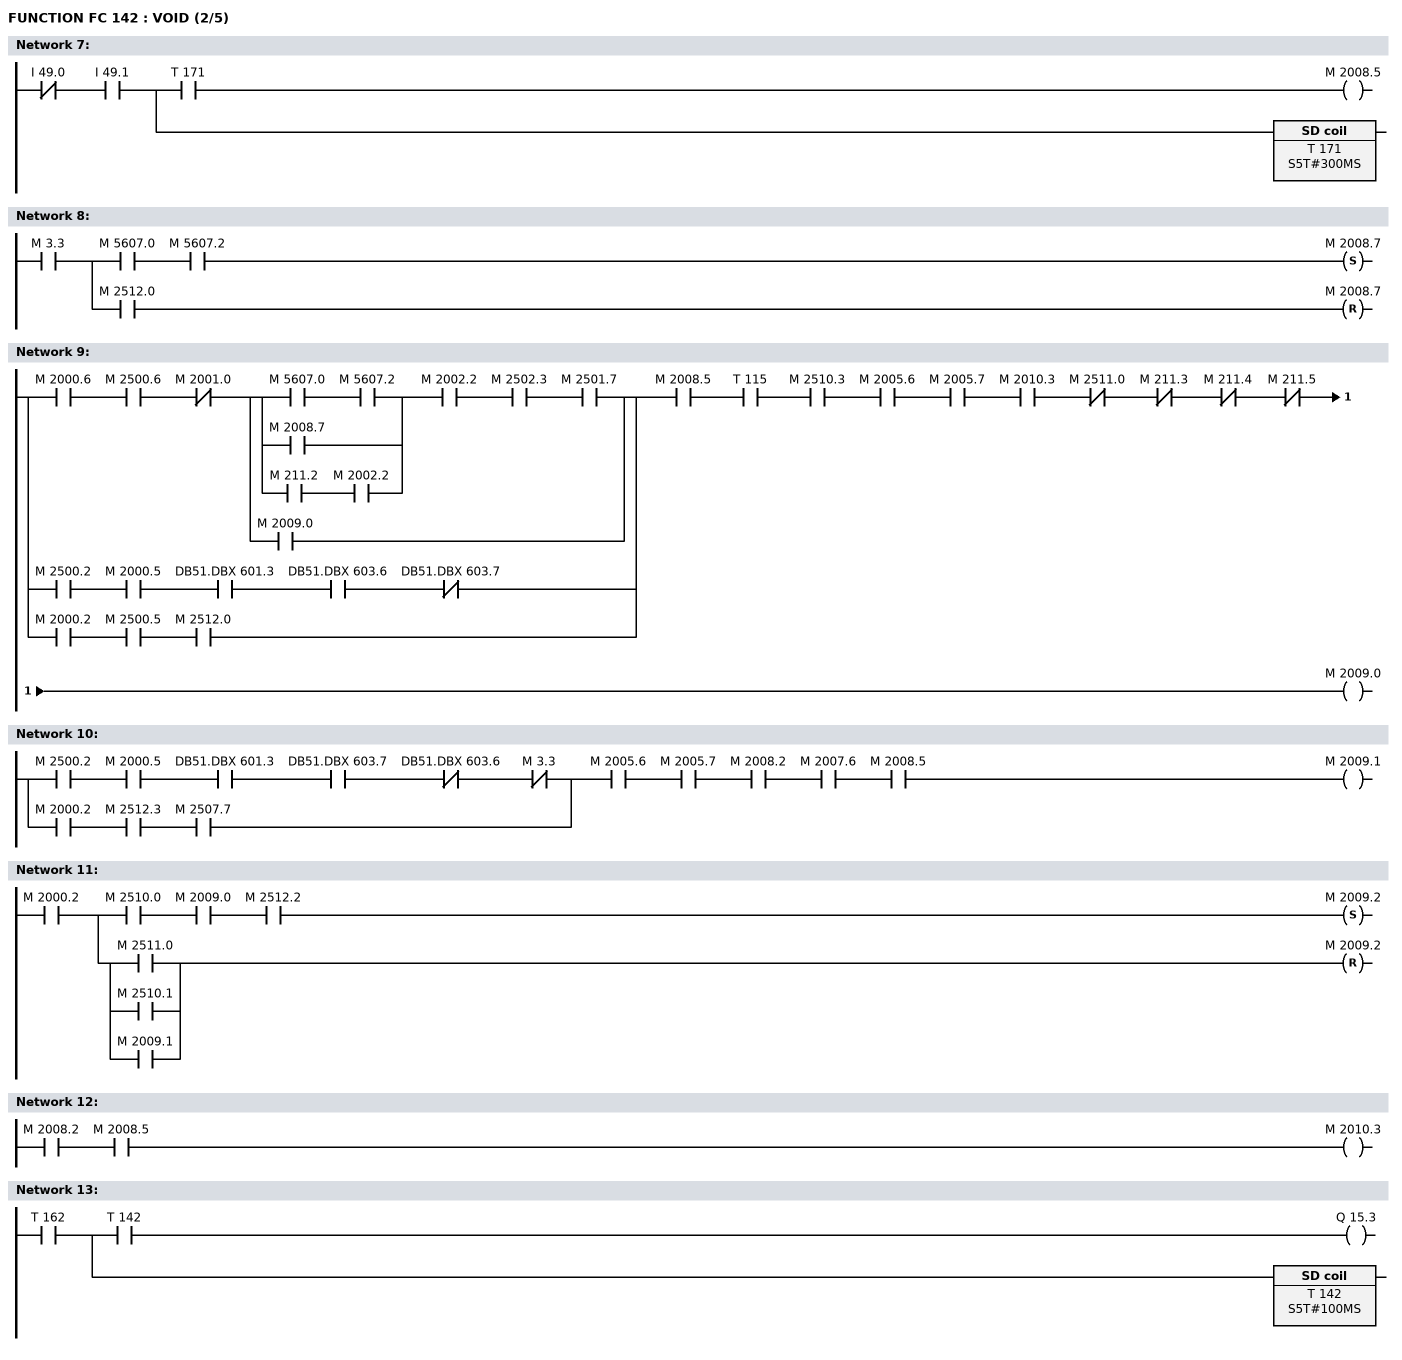

      AN    I     49.0;
      A     I     49.1;
      =     L      0.0;
      A     L      0.0;
      A     T    171;
      =     M   2008.5;
      A     L      0.0;
      BLD   102;
      L     S5T#300MS;
      SD    T    171;
NETWORK
TITLE =

      A     M      3.3;
      =     L      0.0;
      A     L      0.0;
      A     M   5607.0;
      A     M   5607.2;
      S     M   2008.7;
      A     L      0.0;
      A     M   2512.0;
      R     M   2008.7;
NETWORK
TITLE =

      A(    ;
      A     M   2000.6;
      A     M   2500.6;
      AN    M   2001.0;
      A(    ;
      A(    ;
      A     M   5607.0;
      A     M   5607.2;
      O     M   2008.7;
      O     ;
      A     M    211.2;
      A     M   2002.2;
      )     ;
      A     M   2002.2;
      A     M   2502.3;
      A     M   2501.7;
      O     M   2009.0;
      )     ;
      O     ;
      A     M   2500.2;
      A     M   2000.5;
      A     DB51.DBX  601.3;
      A     DB51.DBX  603.6;
      AN    DB51.DBX  603.7;
      O     ;
      A     M   2000.2;
      A     M   2500.5;
      A     M   2512.0;
      )     ;
      A     M   2008.5;
      A     T    115;
      A     M   2510.3;
      A     M   2005.6;
      A     M   2005.7;
      A     M   2010.3;
      AN    M   2511.0;
      AN    M    211.3;
      AN    M    211.4;
      AN    M    211.5;
      =     M   2009.0;
NETWORK
TITLE =

      A(    ;
      A     M   2500.2;
      A     M   2000.5;
      A     DB51.DBX  601.3;
      A     DB51.DBX  603.7;
      AN    DB51.DBX  603.6;
      AN    M      3.3;
      O     ;
      A     M   2000.2;
      A     M   2512.3;
      A     M   2507.7;
      )     ;
      A     M   2005.6;
      A     M   2005.7;
      A     M   2008.2;
      A     M   2007.6;
      A     M   2008.5;
      =     M   2009.1;
NETWORK
TITLE =

      A     M   2000.2;
      =     L      0.0;
      A     L      0.0;
      A     M   2510.0;
      A     M   2009.0;
      A     M   2512.2;
      S     M   2009.2;
      A     L      0.0;
      A(    ;
      O     M   2511.0;
      O     M   2510.1;
      O     M   2009.1;
      )     ;
      R     M   2009.2;
NETWORK
TITLE =

      A     M   2008.2;
      A     M   2008.5;
      =     M   2010.3;
NETWORK
TITLE =

      A     T    162;
      =     L      0.0;
      A     L      0.0;
      A     T    142;
      =     Q     15.3;
      A     L      0.0;
      BLD   102;
      L     S5T#100MS;
      SD    T    142;
NETWORK
TITLE =
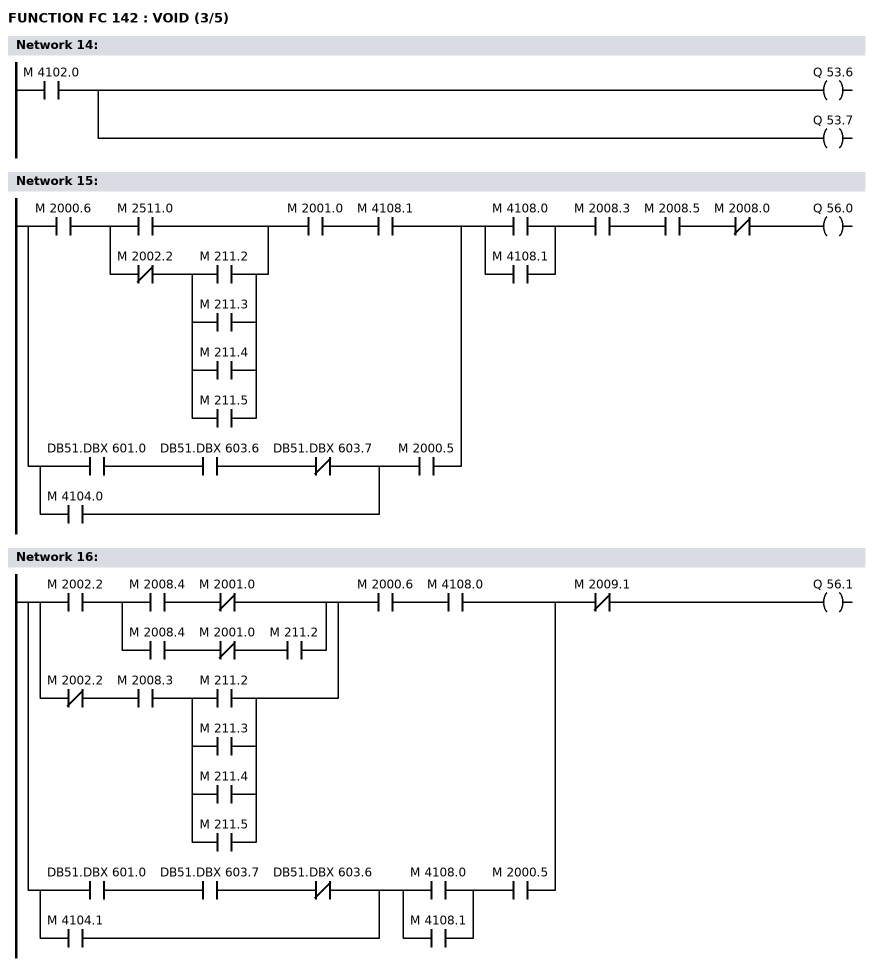

      A     M   4102.0;
      =     Q     53.6;
      =     Q     53.7;
NETWORK
TITLE =

      A(    ;
      A     M   2000.6;
      A(    ;
      O     M   2511.0;
      O     ;
      AN    M   2002.2;
      A(    ;
      O     M    211.2;
      O     M    211.3;
      O     M    211.4;
      O     M    211.5;
      )     ;
      )     ;
      A     M   2001.0;
      A     M   4108.1;
      O     ;
      A(    ;
      A     DB51.DBX  601.0;
      A     DB51.DBX  603.6;
      AN    DB51.DBX  603.7;
      O     M   4104.0;
      )     ;
      A     M   2000.5;
      )     ;
      A(    ;
      O     M   4108.0;
      O     M   4108.1;
      )     ;
      A     M   2008.3;
      A     M   2008.5;
      AN    M   2008.0;
      =     Q     56.0;
NETWORK
TITLE =

      A(    ;
      A(    ;
      A     M   2002.2;
      A(    ;
      A     M   2008.4;
      AN    M   2001.0;
      O     ;
      A     M   2008.4;
      AN    M   2001.0;
      A     M    211.2;
      )     ;
      O     ;
      AN    M   2002.2;
      A     M   2008.3;
      A(    ;
      O     M    211.2;
      O     M    211.3;
      O     M    211.4;
      O     M    211.5;
      )     ;
      )     ;
      A     M   2000.6;
      A     M   4108.0;
      O     ;
      A(    ;
      A     DB51.DBX  601.0;
      A     DB51.DBX  603.7;
      AN    DB51.DBX  603.6;
      O     M   4104.1;
      )     ;
      A(    ;
      O     M   4108.0;
      O     M   4108.1;
      )     ;
      A     M   2000.5;
      )     ;
      AN    M   2009.1;
      =     Q     56.1;
NETWORK
TITLE =
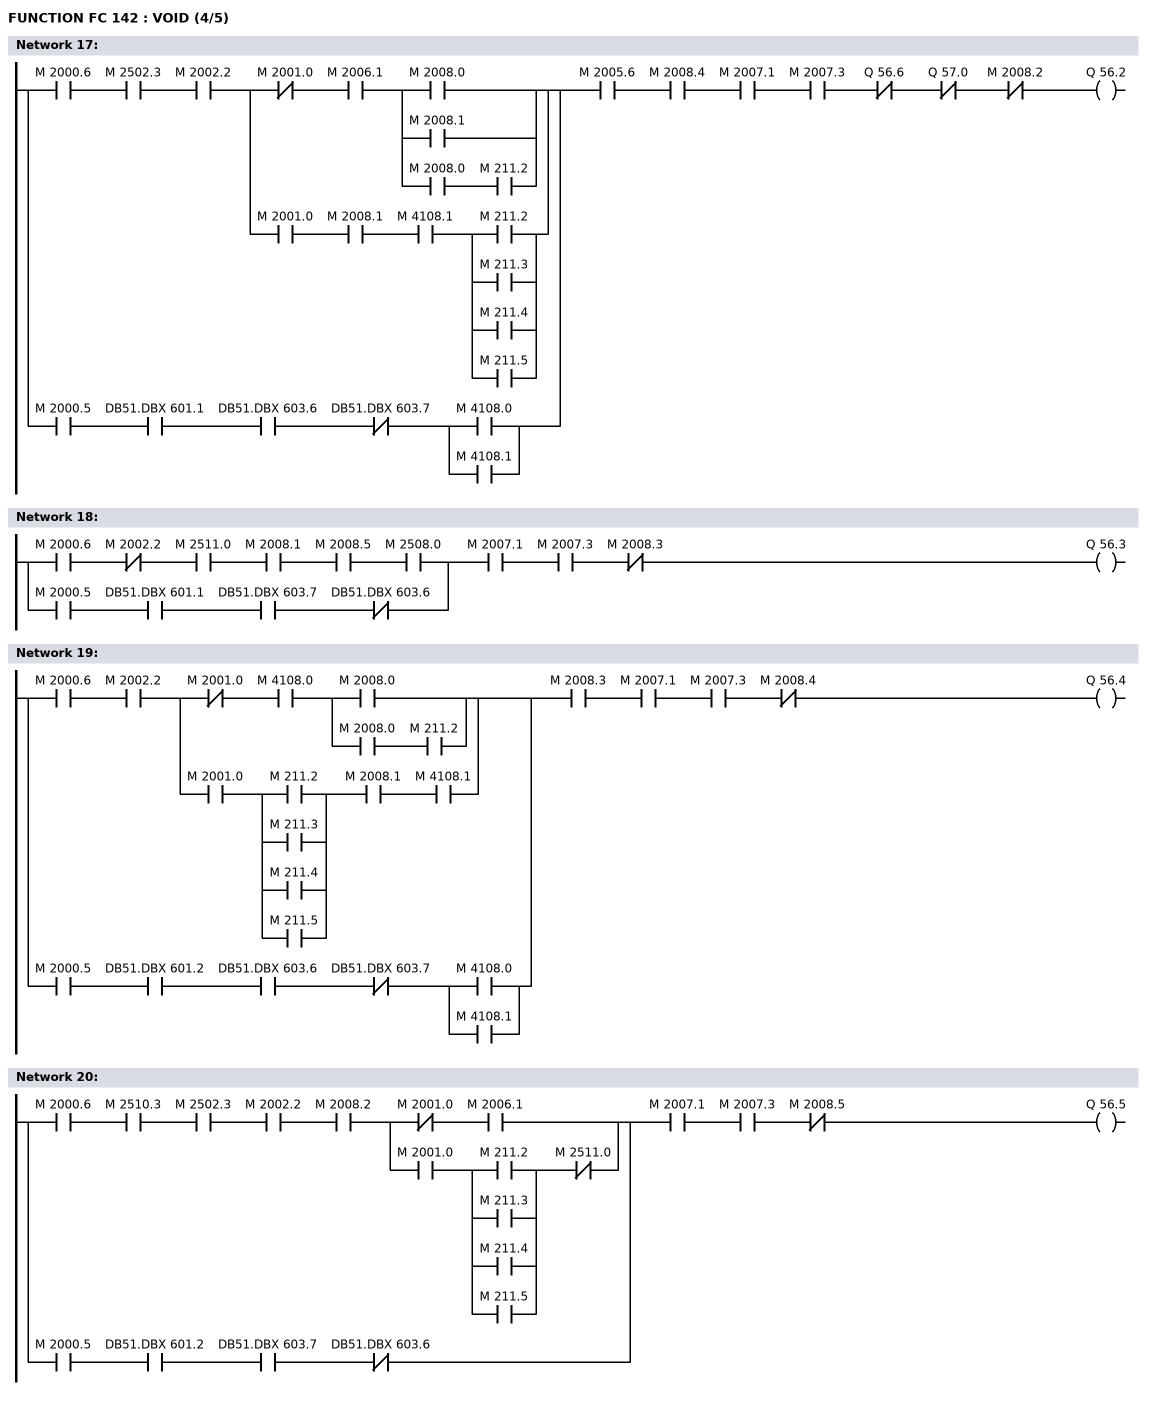

      A(    ;
      A     M   2000.6;
      A     M   2502.3;
      A     M   2002.2;
      A(    ;
      AN    M   2001.0;
      A     M   2006.1;
      A(    ;
      O     M   2008.0;
      O     M   2008.1;
      O     ;
      A     M   2008.0;
      A     M    211.2;
      )     ;
      O     ;
      A     M   2001.0;
      A     M   2008.1;
      A     M   4108.1;
      A(    ;
      O     M    211.2;
      O     M    211.3;
      O     M    211.4;
      O     M    211.5;
      )     ;
      )     ;
      O     ;
      A     M   2000.5;
      A     DB51.DBX  601.1;
      A     DB51.DBX  603.6;
      AN    DB51.DBX  603.7;
      A(    ;
      O     M   4108.0;
      O     M   4108.1;
      )     ;
      )     ;
      A     M   2005.6;
      A     M   2008.4;
      A     M   2007.1;
      A     M   2007.3;
      AN    Q     56.6;
      AN    Q     57.0;
      AN    M   2008.2;
      =     Q     56.2;
NETWORK
TITLE =

      A(    ;
      A     M   2000.6;
      AN    M   2002.2;
      A     M   2511.0;
      A     M   2008.1;
      A     M   2008.5;
      A     M   2508.0;
      O     ;
      A     M   2000.5;
      A     DB51.DBX  601.1;
      A     DB51.DBX  603.7;
      AN    DB51.DBX  603.6;
      )     ;
      A     M   2007.1;
      A     M   2007.3;
      AN    M   2008.3;
      =     Q     56.3;
NETWORK
TITLE =

      A(    ;
      A     M   2000.6;
      A     M   2002.2;
      A(    ;
      AN    M   2001.0;
      A     M   4108.0;
      A(    ;
      O     M   2008.0;
      O     ;
      A     M   2008.0;
      A     M    211.2;
      )     ;
      O     ;
      A     M   2001.0;
      A(    ;
      O     M    211.2;
      O     M    211.3;
      O     M    211.4;
      O     M    211.5;
      )     ;
      A     M   2008.1;
      A     M   4108.1;
      )     ;
      O     ;
      A     M   2000.5;
      A     DB51.DBX  601.2;
      A     DB51.DBX  603.6;
      AN    DB51.DBX  603.7;
      A(    ;
      O     M   4108.0;
      O     M   4108.1;
      )     ;
      )     ;
      A     M   2008.3;
      A     M   2007.1;
      A     M   2007.3;
      AN    M   2008.4;
      =     Q     56.4;
NETWORK
TITLE =

      A(    ;
      A     M   2000.6;
      A     M   2510.3;
      A     M   2502.3;
      A     M   2002.2;
      A     M   2008.2;
      A(    ;
      AN    M   2001.0;
      A     M   2006.1;
      O     ;
      A     M   2001.0;
      A(    ;
      O     M    211.2;
      O     M    211.3;
      O     M    211.4;
      O     M    211.5;
      )     ;
      AN    M   2511.0;
      )     ;
      O     ;
      A     M   2000.5;
      A     DB51.DBX  601.2;
      A     DB51.DBX  603.7;
      AN    DB51.DBX  603.6;
      )     ;
      A     M   2007.1;
      A     M   2007.3;
      AN    M   2008.5;
      =     Q     56.5;
NETWORK
TITLE =
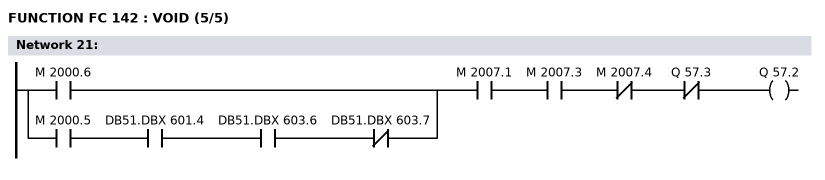

      A(    ;
      O     M   2000.6;
      O     ;
      A     M   2000.5;
      A     DB51.DBX  601.4;
      A     DB51.DBX  603.6;
      AN    DB51.DBX  603.7;
      )     ;
      A     M   2007.1;
      A     M   2007.3;
      AN    M   2007.4;
      AN    Q     57.3;
      =     Q     57.2;
NETWORK
TITLE =

      A     M   2000.5;
      A     DB51.DBX  601.4;
      A     DB51.DBX  603.7;
      AN    DB51.DBX  603.6;
      A     OV;
      A     M   2007.1;
      A     M   2007.3;
      AN    M   2007.5;
      AN    Q     57.2;
      =     Q     57.3;
NETWORK
TITLE =
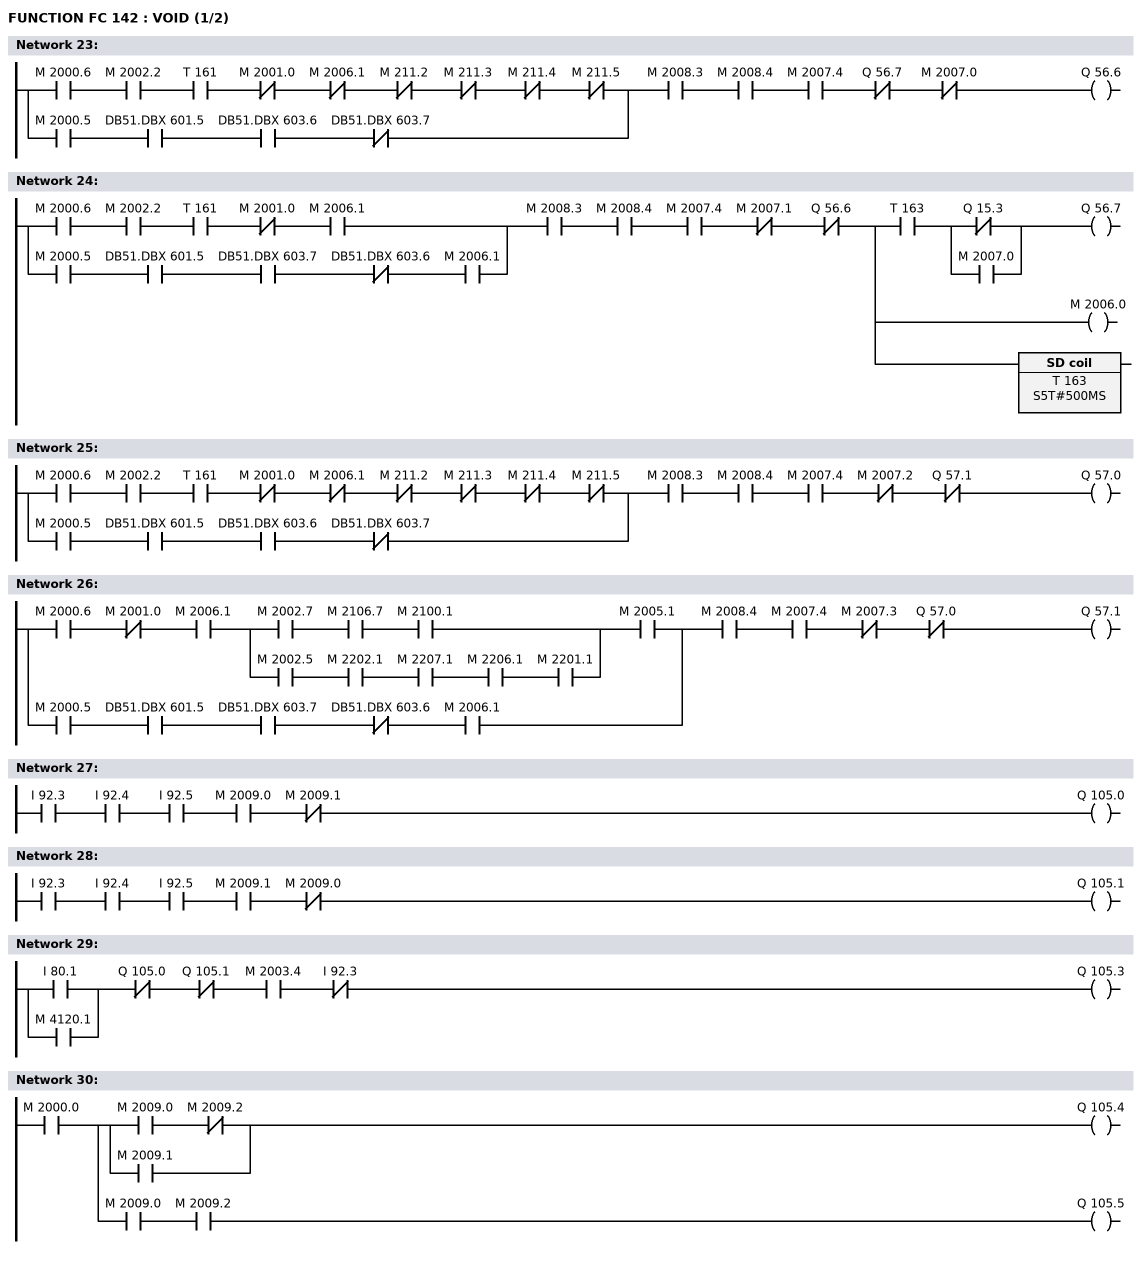

      A(    ;
      A     M   2000.6;
      A     M   2002.2;
      A     T    161;
      AN    M   2001.0;
      AN    M   2006.1;
      AN    M    211.2;
      AN    M    211.3;
      AN    M    211.4;
      AN    M    211.5;
      O     ;
      A     M   2000.5;
      A     DB51.DBX  601.5;
      A     DB51.DBX  603.6;
      AN    DB51.DBX  603.7;
      )     ;
      A     M   2008.3;
      A     M   2008.4;
      A     M   2007.4;
      AN    Q     56.7;
      AN    M   2007.0;
      =     Q     56.6;
NETWORK
TITLE =

      A(    ;
      A     M   2000.6;
      A     M   2002.2;
      A     T    161;
      AN    M   2001.0;
      A     M   2006.1;
      O     ;
      A     M   2000.5;
      A     DB51.DBX  601.5;
      A     DB51.DBX  603.7;
      AN    DB51.DBX  603.6;
      A     M   2006.1;
      )     ;
      A     M   2008.3;
      A     M   2008.4;
      A     M   2007.4;
      AN    M   2007.1;
      AN    Q     56.6;
      =     L      0.0;
      A     L      0.0;
      A     T    163;
      A(    ;
      ON    Q     15.3;
      O     M   2007.0;
      )     ;
      =     Q     56.7;
      A     L      0.0;
      BLD   102;
      =     M   2006.0;
      A     L      0.0;
      BLD   102;
      L     S5T#500MS;
      SD    T    163;
NETWORK
TITLE =

      A(    ;
      A     M   2000.6;
      A     M   2002.2;
      A     T    161;
      AN    M   2001.0;
      AN    M   2006.1;
      AN    M    211.2;
      AN    M    211.3;
      AN    M    211.4;
      AN    M    211.5;
      O     ;
      A     M   2000.5;
      A     DB51.DBX  601.5;
      A     DB51.DBX  603.6;
      AN    DB51.DBX  603.7;
      )     ;
      A     M   2008.3;
      A     M   2008.4;
      A     M   2007.4;
      AN    M   2007.2;
      AN    Q     57.1;
      =     Q     57.0;
NETWORK
TITLE =

      A(    ;
      A     M   2000.6;
      AN    M   2001.0;
      A     M   2006.1;
      A(    ;
      A     M   2002.7;
      A     M   2106.7;
      A     M   2100.1;
      O     ;
      A     M   2002.5;
      A     M   2202.1;
      A     M   2207.1;
      A     M   2206.1;
      A     M   2201.1;
      )     ;
      A     M   2005.1;
      O     ;
      A     M   2000.5;
      A     DB51.DBX  601.5;
      A     DB51.DBX  603.7;
      AN    DB51.DBX  603.6;
      A     M   2006.1;
      )     ;
      A     M   2008.4;
      A     M   2007.4;
      AN    M   2007.3;
      AN    Q     57.0;
      =     Q     57.1;
NETWORK
TITLE =

      A     I     92.3;
      A     I     92.4;
      A     I     92.5;
      A     M   2009.0;
      AN    M   2009.1;
      =     Q    105.0;
NETWORK
TITLE =

      A     I     92.3;
      A     I     92.4;
      A     I     92.5;
      A     M   2009.1;
      AN    M   2009.0;
      =     Q    105.1;
NETWORK
TITLE =

      A(    ;
      O     I     80.1;
      O     M   4120.1;
      )     ;
      AN    Q    105.0;
      AN    Q    105.1;
      A     M   2003.4;
      AN    I     92.3;
      =     Q    105.3;
NETWORK
TITLE =

      A     M   2000.0;
      =     L      0.0;
      A     L      0.0;
      A(    ;
      A     M   2009.0;
      AN    M   2009.2;
      O     M   2009.1;
      )     ;
      =     Q    105.4;
      A     L      0.0;
      A     M   2009.0;
      A     M   2009.2;
      =     Q    105.5;
NETWORK
TITLE =
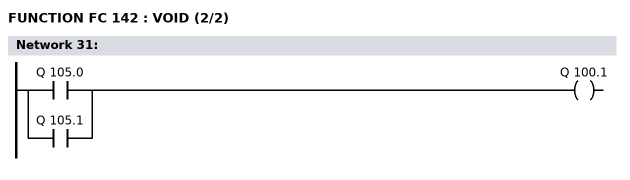

      O     Q    105.0;
      O     Q    105.1;
      =     Q    100.1;
END_FUNCTION

FUNCTION_BLOCK FB 143
TITLE =
VERSION : 0.1


VAR
  S708_LM_DC_PIN : FB 424;
  S708_LM_DC_1ST_CLAMP1 : FB 424;
  S708_LM_DC_1ST_CLAMP2 : FB 424;
  S708_LM_DC_1ST_CLAMP3 : FB 424;
  S708_LM_DC_1ST_CLAMP4 : FB 424;
  S708_LM_DC_2ND_CLAMP1 : FB 424;
  S708_LM_DC_2ND_CLAMP2 : FB 424;
  S708_LM_DC_2ND_CLAMP3 : FB 424;
  S708_LM_DC_2ND_CLAMP4 : FB 424;
  S708_LM_DC_2ND_CLAMP5 : FB 424;
  S708_LM_DC_STK_PIN : FB 424;
  S708_LM_DC_OTR_CLAMP : FB 424;
  S708_LM_DC_ASSY_CLAMP : FB 424;
  S708_LM_DC_FF_PIN : FB 424;
  S708_LM_DC_FF_CLAMP : FB 424;
  S708_LM_DC_2ND_CLAMP6 : FB 424;
  S708_LM_DC_2ND_CLAMP7 : FB 424;
  S708_LM_DC_1ST_CLAMP5 : FB 424;
END_VAR
BEGIN
NETWORK
TITLE =
